VAR_IN_OUT PERSISTENT
	DsStnSeqRepCall : DSV2_fbStationSequenceRecipeCall;
	DsStnSubRepCall : DS_fbStationSubRecipeCall;
	DsBasketInfo : DSV2_BasketInfo;
END_VAR

VAR_OUTPUT PERSISTENT
	bProcessCompleted : BOOL;
	bProcessInProgressFlag : BOOL;
	bProcessHaltFlag: BOOL;
	bCallStnSeqRecipeErr: BOOL;
	bInvalidProcessStepErr: BOOL;
	DSStnSeqProOutput :DS_StnSeqProOutput;
	iCurrentProcessStep : INT;
	iComConProcessTimeEV: INT;
	ARiCurrentCycle : ARRAY [1..10] OF INT;
	iCurrentProcessTime : INT; (*Total Process Time Since Start*)
	iPreviousProcessTime : INT; (*Total Process Time - Previous process*)
	iStnSeqProcessCase: INT; (* Temporary - Will transfer to Var_Persistent later*)

END_VAR
VAR
(*	DsBufferSubRecipeMemory : Ds_SubRecipeMemory;
	bCallStnSeqSubProCompleted : BOOL;
	bCallStnSeqRepErr : BOOL;
	bCallStnSubRepErr : BOOL;
*)	rebProcessStart: R_TRIG;


	bCallStnSeqSubProEn: BOOL;

	bStCon7BelowTargetVacuumLevel : BOOL;
	bStCon8AboveTargetVacuumLevel : BOOL;
	bStCon9BelowTargetPressureLevel : BOOL;
	bStCon10AboveTargetPressureLevel : BOOL;
	bStCon11BelowTargetProTankTempLevel : BOOL;
	bStCon12AboveTargetProTankTempLevel : BOOL;
	bStCon13BelowTargetSubTankTempLevel : BOOL;
	bStCon14AboveTargetSubTankTempLevel : BOOL;

	bComCon7BelowTargetVacuumLevel : BOOL;
	bComCon8AboveTargetVacuumLevel : BOOL;
	bComCon9BelowTargetPressureLevel : BOOL;
	bComCon10AboveTargetPressureLevel : BOOL;
	bComCon11BelowTargetProTankTempLevel : BOOL;
	bComCon12AboveTargetProTankTempLevel : BOOL;
	bComCon13BelowTargetSubTankTempLevel : BOOL;
	bComCon14AboveTargetSubTankTempLevel : BOOL;

	tProcess1secClockPulse: TON;
	retProcess1secClockPulse: R_TRIG;
	rebProcessCompleted: R_TRIG;
	ClearFL: INT;
	iCurrentProcessStepBuffer: INT;
	rebInvalidProcessStepErr: R_TRIG;
	rebStnSeqSubCallCompleted: R_TRIG;
	rebCallStnSeqRecipeErr: R_TRIG;
	rebCallStnSubRecipeErr: R_TRIG;
	tStartProcess1secClockPulse: TON;
	retStartProcess1secClockPulse: R_TRIG;
	bTempCallCompleted: BOOL;
	bTempInvalidProcessStepErr: BOOL;
	bTempCallStnSeqRecipeErr: BOOL;
	bTempCallStnSubRecipeErr: BOOL;
	sTempsSubDescription: STRING(50);
	DsTempSubRecipeMemory: DS_SubRecipeMemory;
	iTempSeqStep: INT;
	bTempInvalidProcessStepErrPls: BOOL;
	rebProcessHalt: R_TRIG;
	febProcessHalt: F_TRIG;
END_VAR

VAR PERSISTENT
	StationfbCallStnSeqSubPro: fbCallStnSeqSubPro;
	bStartConditionPassed: BOOL;
	bCompleteConditionPassed: BOOL;
	bStationProcessTimerComplete: BOOL;
	iComConProcessTime: INT;

END_VAR

VAR_OUTPUT
END_VAR
*)

(*Temporary - Create Total Process Time SV *)
iTPTFL := 1;
bEndStep:= FALSE;

	FOR iTPTFL := 1 TO IStationSubRecipeArrayQty DO
		IF
		fbStationSequenceRecipefb.ARDsStorageStationSequenceRecipeMemory[DsBasketInfo.iStationSeqenceRecipeNo].AR10iStationSubProNo[iTPTFL] > 0
		AND
		fbStationSequenceRecipefb.ARDsStorageStationSequenceRecipeMemory[DsBasketInfo.iStationSeqenceRecipeNo].AR10iStationSubProNo[iTPTFL] <= IStationSubRecipeArrayQty
		AND NOT
		bEndStep
		THEN
		ARiTotalTimeSV[iTPTFL] := fbStationSubRecipefb.ARDsStorageSubRecipeMemory[(**)fbStationSequenceRecipefb.ARDsStorageStationSequenceRecipeMemory[DsBasketInfo.iStationSeqenceRecipeNo].AR10iStationSubProNo[iTPTFL](**)].iComCon5ProcessTimer;
		ELSE
		bEndStep := TRUE;
		ARiTotalTimeSV[iTPTFL] := 0;
		END_IF
	END_FOR
DsBasketInfo.iStationSeqenceRecipeNo;


iTotalProcessTimeSV :=
ARiTotalTimeSV[1] +
ARiTotalTimeSV[2] +
ARiTotalTimeSV[3] +
ARiTotalTimeSV[4] +
ARiTotalTimeSV[5] +
ARiTotalTimeSV[6] +
ARiTotalTimeSV[7] +
ARiTotalTimeSV[8] +
ARiTotalTimeSV[9] +
ARiTotalTimeSV[10];


IF bProcessInProgressFlag AND NOT bProcessHalt AND retStartProcess1secClockPulse.Q  THEN
iTotalProcessTimeEVInt := iTotalProcessTimeEVInt+1;
END_IF

IF (bProcessInProgressFlag OR bProcessHalt OR bProcessCompleted) AND NOT bProcessHalt AND iTotalProcessTimeSV - iTotalProcessTimeEVInt > 0 THEN
iTotalProcessTimeEV := iTotalProcessTimeSV - iTotalProcessTimeEVInt;
END_IF

IF (bProcessInProgressFlag OR bProcessHalt OR bProcessCompleted) AND NOT bProcessHalt AND iTotalProcessTimeSV - iTotalProcessTimeEVInt <= 0 THEN
iTotalProcessTimeEV := 0;
END_IF

IF NOT bProcessInProgressFlag AND NOT  bProcessHalt AND NOT bProcessCompleted THEN
iTotalProcessTimeEV := iTotalProcessTimeSV;
END_IF






(*Temp Create to generate total time for Loaded In Basket. Used in Time Optimisation*)
iCallTotalTimeMFL := 1;
iCallTotalTimeSFL := 1;

IF iCallTotalTimeMFL >0 AND iCallTotalTimeMFL < 5+1 THEN

	FOR iCallTotalTimeMFL := 1 TO 5 DO

		iCallTotalTimeSFL := 1;
		bCallTotalTimeEndStep:= FALSE;

		IF iCallTotalTimeSFL >0 AND iCallTotalTimeSFL < IStationSubRecipeArrayQty+1 THEN
			FOR iCallTotalTimeSFL := 1 TO IStationSubRecipeArrayQty DO
				IF
				fbStationSequenceRecipefb.ARDsStorageStationSequenceRecipeMemory[AR5iCallTotalTimeRecipeNo[iCallTotalTimeMFL]].AR10iStationSubProNo[iCallTotalTimeSFL] > 0
				AND
				fbStationSequenceRecipefb.ARDsStorageStationSequenceRecipeMemory[AR5iCallTotalTimeRecipeNo[iCallTotalTimeMFL]].AR10iStationSubProNo[iCallTotalTimeSFL] <= IStationSubRecipeArrayQty
				AND NOT
				bCallTotalTimeEndStep
				THEN
				AR2SiTimeOptimiseTotalTimeSV[iCallTotalTimeMFL,iCallTotalTimeSFL] := fbStationSubRecipefb.ARDsStorageSubRecipeMemory[(**)fbStationSequenceRecipefb.ARDsStorageStationSequenceRecipeMemory[AR5iCallTotalTimeRecipeNo[iCallTotalTimeMFL]].AR10iStationSubProNo[iCallTotalTimeSFL](**)].iComCon5ProcessTimer;
				ELSE
				bCallTotalTimeEndStep := TRUE;
				AR2SiTimeOptimiseTotalTimeSV[iCallTotalTimeMFL,iCallTotalTimeSFL] := 0;
				END_IF
			END_FOR
		END_IF
	END_FOR
END_IF

iCalculateMFL := 1;


IF iCalculateMFL >0 AND iCalculateMFL < 5+1 THEN

	FOR iCalculateMFL := 1 TO 5 DO

		AR5iCalledTotalProcessTimeSV[iCalculateMFL] :=
		AR2SiTimeOptimiseTotalTimeSV[iCalculateMFL,1] +
		AR2SiTimeOptimiseTotalTimeSV[iCalculateMFL,2] +
		AR2SiTimeOptimiseTotalTimeSV[iCalculateMFL,3] +
		AR2SiTimeOptimiseTotalTimeSV[iCalculateMFL,4] +
		AR2SiTimeOptimiseTotalTimeSV[iCalculateMFL,5] +
		AR2SiTimeOptimiseTotalTimeSV[iCalculateMFL,6] +
		AR2SiTimeOptimiseTotalTimeSV[iCalculateMFL,7] +
		AR2SiTimeOptimiseTotalTimeSV[iCalculateMFL,8] +
		AR2SiTimeOptimiseTotalTimeSV[iCalculateMFL,9] +
		AR2SiTimeOptimiseTotalTimeSV[iCalculateMFL,10];
		
	END_FOR
END_IF


(*[][][][][][][][][][][][][][][][][][][][][][][][][][][][][][][][][][][][][][][][][][][][][][][][][][][][][][][][][][][][][][][][][][][][][][][][]-Group in StationSequnceRecipe and StationSubRecipe-[][][][][][][][][][][][][][][][][][][][][][][][][][][][][][][][][][][][][][][][][][][][][][][][][][][][][][][][][][][][][][][][][][][][][][][][]*)
fbStationSequenceRecipefb(
	bSavePB								:=bSavePB ,
	bLoadPB								:=bLoadPB ,
	bClearPB							:=bClearPB_SSER ,
	bCopyPB								:=DsStnSeqRepStore.bCopyPB ,
	iCopyToSubRecipeNo						:=DsStnSeqRepStore.iCopyToSubRecipeNo ,
	iStnID									:=iCurrentStationAddress ,
	iStationSequenceRecipeNo				:=DsStnSeqRepStore.iStationSequenceRecipeNo ,
	sStationSequenceRecipeDescription			:=DsStnSeqRepStore.sStationSequenceRecipeDescription ,
	DsInStationSequenceRecipeMemory			:=DsStnSeqRepStore.DsStationSequenceRecipeMemory ,
	ARDsSSERSourceMinMaxTime_Uni			:=ARDsSSERSourceMinMaxTime_Uni ,
	Call_iStationSequenceRecipe				:=DsStnSeqRepCall.Call_iStationSequenceRecipe ,
	bCallPB									:=DsStnSeqRepCall.bCallPB ,
	bSaveInd								=>bSaveInd ,
	bLoadInd								=>bLoadInd ,
	bClearInd								=>bClearInd_SSUR ,
	bCallCompleted							=>DsStnSeqRepCall.bCallCompleted ,
	bInvalidCallStationSequenceNoHold			=>DsStnSeqRepCall.bInvalidCallStationSequenceNoHold ,
	bInvalidCallStationSequenceNoPulse		=>DsStnSeqRepCall.bInvalidCallStationSequenceNoPulse ,
	Call_sSequenceRecipeDescription			=>DsStnSeqRepCall.Call_sSequenceRecipeDescription ,
	Call_DsStationSequenceRecipeMemory		=>DsStnSeqRepCall.Call_DsStationSequenceRecipeMemory );

	

	
	
(*

fbStationSequenceRecipefb(
	bSavePB:=bSavePB ,
	bLoadPB:=bLoadPB ,
	bCopyPB:=DsStnSeqRepStore.bCopyPB ,
	iCopyToSubRecipeNo:= DsStnSeqRepStore.iCopyToSubRecipeNo,
	iStationSequenceRecipeNo:=DsStnSeqRepStore.iStationSequenceRecipeNo ,
	sStationSequenceRecipeDescription:=DsStnSeqRepStore.sStationSequenceRecipeDescription ,
	DsInStationSequenceRecipeMemory:=DsStnSeqRepStore.DsStationSequenceRecipeMemory ,
	Call_iStationSequenceRecipe:= DsStnSeqRepCall.Call_iStationSequenceRecipe,
	bCallPB:=DsStnSeqRepCall.bCallPB ,
	bSaveInd=>bSaveInd ,
	bLoadInd=>bLoadInd ,
	bCallCompleted=>DsStnSeqRepCall.bCallCompleted ,
	bInvalidCallStationSequenceNoHold=>DsStnSeqRepCall.bInvalidCallStationSequenceNoHold ,
	bInvalidCallStationSequenceNoPulse=>DsStnSeqRepCall.bInvalidCallStationSequenceNoPulse ,
	Call_sSequenceRecipeDescription=>DsStnSeqRepCall.Call_sSequenceRecipeDescription ,
	Call_DsStationSequenceRecipeMemory=>DsStnSeqRepCall.Call_DsStationSequenceRecipeMemory );
*)
fbStationSubRecipefb(
	bSavePB:= bSavePB,
	bLoadPB := bLoadPB,
	bClearPB:= bClearPB_SSUR,
	bCopyPB:=DsStnSubRepStore.bCopyPB ,
	iCopyToSubRecipeNo:= DsStnSubRepStore.iCopyToSubRecipeNo,
	DsStnSeqProInput:= DsStnSeqProInput,
	iSubRecipeNo:= DsStnSubRepStore.iSubRecipeNo,
	sSubRecipeDescription:= DsStnSubRepStore.sSubRecipeDescription,
	DsInSubRecipeMemory:= DsStnSubRepStore.DsSubRecipeMemory,
	Call_iSubRecipe:= DsStnSubRepCall.Call_iSubRecipe,
	bCallPB:= DsStnSubRepCall.bCallPB,
	bSaveInd=>bSaveInd ,
	bLoadInd=>bLoadInd ,
	bClearInd=>bClearInd_SSUR,
	bCallCompleted=> DsStnSubRepCall.bCallCompleted,
	bInvalidCallSubRecipeNoHold=> DsStnSubRepCall.bInvalidCallSubRecipeNoHold,
	bInvalidCallSubRecipeNoPulse=> DsStnSubRepCall.bInvalidCallSubRecipeNoPulse,
	Call_sSubDescription=> DsStnSubRepCall.Call_sSubDescription,
	Call_DsSubRecipeMemory=> DsStnSubRepCall.Call_DsSubRecipeMemory);


(*[][][][][][][][][][][][][][][][][][][][][][][][][][][][][][][][][][][][][][][][][][][][][][][][][][][][][][][][][][][][][][][][][][][][][][][][]-Only FB StnSeqProcess-[][][][][][][][][][][][][][][][][][][][][][][][][][][][][][][][][][][][][][][][][][][][][][][][][][][][][][][][][][][][][][][][][][][][][][][][]*)

(*[][][][][][][][][][][][][][][][][][]-Generate Current Process Time-[][][][][][][][][][][][][][][][][][]*)
tProcess1secClockPulse(IN:=(bProcessInProgressFlag OR bProcessCompleted) AND NOT tProcess1secClockPulse.Q , PT:= T#1s, Q=> , ET=> );
retProcess1secClockPulse(CLK:=tProcess1secClockPulse.Q , Q=> );

IF bProcessInProgressFlag AND NOT bProcessHalt AND retProcess1secClockPulse.Q THEN
iCurrentProcessTime := iCurrentProcessTime+1;
END_IF


IF (bProcessInProgressFlag OR bProcessCompleted OR bOutputCutOffEn) AND NOT bProcessHalt AND retProcess1secClockPulse.Q THEN
iNonStopCurrentProcessTime := iNonStopCurrentProcessTime+1;
END_IF


(*[][][][][][][][][][][][][][][][][][]-Complete Condition Process Time Handling-[][][][][][][][][][][][][][][][][][]*)

(*Generate CompleteCondition Process Time Elapse Value (Reverse Counting)*)
IF bProcessInProgressFlag AND NOT bProcessHalt AND StationfbCallStnSeqSubPro.BufferDsSubRecipeMemory.bComCon20EnProcessTimer AND iStnSeqProcessCaseNo = 3 THEN
iComConProcessTimeEV := StationfbCallStnSeqSubPro.BufferDsSubRecipeMemory.iComCon5ProcessTimer - iComConProcessTime;
END_IF

IF (NOT bProcessInProgressFlag AND NOT bProcessHalt) OR NOT StationfbCallStnSeqSubPro.BufferDsSubRecipeMemory.bComCon20EnProcessTimer OR iStnSeqProcessCaseNo <> 3 THEN
iComConProcessTimeEV := 0;
END_IF



(*Start Complete Condition Timer If Available*)
tStartProcess1secClockPulse(IN:=StationfbCallStnSeqSubPro.BufferDsSubRecipeMemory.bComCon20EnProcessTimer AND NOT tStartProcess1secClockPulse.Q AND iStnSeqProcessCaseNo = 3 , PT:=T#1s , Q=> , ET=> );
retStartProcess1secClockPulse(CLK:=tStartProcess1secClockPulse.Q , Q=> );

IF bProcessInProgressFlag AND NOT bProcessHalt AND retStartProcess1secClockPulse.Q  THEN
iComConProcessTime := iComConProcessTime+1;
END_IF

IF bProcessInProgressFlag AND NOT bProcessHalt AND iComConProcessTime >= StationfbCallStnSeqSubPro.BufferDsSubRecipeMemory.iComCon5ProcessTimer THEN
bStationProcessTimerComplete := TRUE;
ELSE
bStationProcessTimerComplete := FALSE;
END_IF


(*[][][][][][][][][][][][][][][][][][]-Generate Above/Below-Start Condition-[][][][][][][][][][][][][][][][][][]*)

IF DsStnSeqProInput.iVacuumLevelPV < StationfbCallStnSeqSubPro.BufferDsSubRecipeMemory.iStCon1TargetVacuumLevel THEN
bStCon11BelowTargetVacuumLevel := TRUE;
ELSE
bStCon11BelowTargetVacuumLevel := FALSE;
END_IF

IF DsStnSeqProInput.iVacuumLevelPV >= StationfbCallStnSeqSubPro.BufferDsSubRecipeMemory.iStCon1TargetVacuumLevel THEN
bStCon12AboveTargetVacuumLevel := TRUE;
ELSE
bStCon12AboveTargetVacuumLevel := FALSE;
END_IF

IF DsStnSeqProInput.iPressureLevelPV < StationfbCallStnSeqSubPro.BufferDsSubRecipeMemory.iStCon2TargetPressureLevel THEN
bStCon13BelowTargetPressureLevel := TRUE;
ELSE
bStCon13BelowTargetPressureLevel := FALSE;
END_IF

IF DsStnSeqProInput.iPressureLevelPV >= StationfbCallStnSeqSubPro.BufferDsSubRecipeMemory.iStCon2TargetPressureLevel THEN
bStCon14AboveTargetPressureLevel := TRUE;
ELSE
bStCon14AboveTargetPressureLevel := FALSE;
END_IF

IF DsStnSeqProInput.iProTankTempLevelPV < StationfbCallStnSeqSubPro.BufferDsSubRecipeMemory.iStCon3TargetProTankTempLevel THEN
bStCon15BelowTargetProTankTempLevel := TRUE;
ELSE
bStCon15BelowTargetProTankTempLevel := FALSE;
END_IF

IF DsStnSeqProInput.iProTankTempLevelPV >= StationfbCallStnSeqSubPro.BufferDsSubRecipeMemory.iStCon3TargetProTankTempLevel THEN
bStCon16AboveTargetProTankTempLevel := TRUE;
ELSE
bStCon16AboveTargetProTankTempLevel := FALSE;
END_IF

IF DsStnSeqProInput.iSubTankTempLevelPV < StationfbCallStnSeqSubPro.BufferDsSubRecipeMemory.iStCon4TargetSubTankTempLevel THEN
bStCon17BelowTargetSubTankTempLevel := TRUE;
ELSE
bStCon17BelowTargetSubTankTempLevel := FALSE;
END_IF

IF DsStnSeqProInput.iSubTankTempLevelPV >= StationfbCallStnSeqSubPro.BufferDsSubRecipeMemory.iStCon4TargetSubTankTempLevel THEN
bStCon18AboveTargetSubTankTempLevel := TRUE;
ELSE
bStCon18AboveTargetSubTankTempLevel := FALSE;
END_IF


(*[][][][][][][][][][][][][][][][][][]-Generate Above/Below-Complete Condition-[][][][][][][][][][][][][][][][][][]*)

IF DsStnSeqProInput.iVacuumLevelPV < StationfbCallStnSeqSubPro.BufferDsSubRecipeMemory.iComCon1TargetVacuumLevel THEN
bComCon11BelowTargetVacuumLevel := TRUE;
ELSE
bComCon11BelowTargetVacuumLevel := FALSE;
END_IF

IF DsStnSeqProInput.iVacuumLevelPV >= StationfbCallStnSeqSubPro.BufferDsSubRecipeMemory.iComCon1TargetVacuumLevel THEN
bComCon12AboveTargetVacuumLevel := TRUE;
ELSE
bComCon12AboveTargetVacuumLevel := FALSE;
END_IF

IF DsStnSeqProInput.iPressureLevelPV < StationfbCallStnSeqSubPro.BufferDsSubRecipeMemory.iComCon2TargetPressureLevel THEN
bComCon13BelowTargetPressureLevel := TRUE;
ELSE
bComCon13BelowTargetPressureLevel := FALSE;
END_IF

IF DsStnSeqProInput.iPressureLevelPV >= StationfbCallStnSeqSubPro.BufferDsSubRecipeMemory.iComCon2TargetPressureLevel THEN
bComCon14AboveTargetPressureLevel := TRUE;
ELSE
bComCon14AboveTargetPressureLevel := FALSE;
END_IF

IF DsStnSeqProInput.iProTankTempLevelPV < StationfbCallStnSeqSubPro.BufferDsSubRecipeMemory.iComCon3TargetProTankTempLevel THEN
bComCon15BelowTargetProTankTempLevel := TRUE;
ELSE
bComCon15BelowTargetProTankTempLevel := FALSE;
END_IF

IF DsStnSeqProInput.iProTankTempLevelPV >= StationfbCallStnSeqSubPro.BufferDsSubRecipeMemory.iComCon3TargetProTankTempLevel THEN
bComCon16AboveTargetProTankTempLevel := TRUE;
ELSE
bComCon16AboveTargetProTankTempLevel := FALSE;
END_IF

IF DsStnSeqProInput.iSubTankTempLevelPV < StationfbCallStnSeqSubPro.BufferDsSubRecipeMemory.iComCon4TargetSubTankTempLevel THEN
bComCon17BelowTargetSubTankTempLevel := TRUE;
ELSE
bComCon17BelowTargetSubTankTempLevel := FALSE;
END_IF

IF DsStnSeqProInput.iSubTankTempLevelPV >= StationfbCallStnSeqSubPro.BufferDsSubRecipeMemory.iComCon4TargetSubTankTempLevel THEN
bComCon18AboveTargetSubTankTempLevel := TRUE;
ELSE
bComCon18AboveTargetSubTankTempLevel := FALSE;
END_IF

(*[][][][][][][][][][][][][][][][][][]-General-[][][][][][][][][][][][][][][][][][]*)
rebProcessHalt(CLK:=bProcessHalt , Q=> );

febProcessHalt(CLK:=bProcessHalt , Q=> );

IF rebProcessHalt.Q AND bProcessInProgressFlag THEN
bProcessInProgressFlag := FALSE;
bProcessHaltFlag := TRUE;
END_IF

IF febProcessHalt.Q AND bProcessHaltFlag THEN
bProcessInProgressFlag := TRUE;
bProcessHaltFlag := FALSE;
END_IF



IF bProcessReset OR NOT DsBasketInfo.bAvailibility THEN
bProcessInProgressFlag := FALSE;
bCallStnSeqRecipeErr := FALSE;
bInvalidProcessStepErr := FALSE;
bCallStnSeqSubProEn := FALSE;
bProcessCompleted := FALSE;
bProcessHaltFlag := FALSE;

iStnSeqProcessCaseNo := 0;
iCurrentProcessStep := 0;
iCurrentProcessTime := 0;
iNonStopCurrentProcessTime := 0;
(*iTotalProcessTimeEV:=0;*)
iTotalProcessTimeEVInt := 0;
iComConProcessTime := 0;
iTotalProcessTimeEV := 0; (*Add New*)
DsStnSeqRepCall:=DsStnSeqRepCallEmpty;
DsStnSubRepCall:=DsStnSubRepCallEmpty;
ClearFL := 1;

	FOR ClearFL := 1 TO IStationSubRecipeArrayQty(*10*) DO
		ARiCurrentCycle[ClearFL] := 0;
	END_FOR

END_IF




rebProcessStart(CLK:=bProcessStart  , Q=> );

IF rebProcessStart.Q AND NOT bProcessHaltFlag AND NOT bProcessInProgressFlag AND NOT bProcessCompleted THEN
iStnSeqProcessCaseNo := 1;
iCurrentProcessStep := 1;
ARiCurrentCycle[iCurrentProcessStep] := 1;
bProcessInProgressFlag := TRUE;
END_IF


(*[][][][][][][][][][][][][][][][][][]-FB Declaration-[][][][][][][][][][][][][][][][][][]*)

StationfbCallStnSeqSubPro(
	bCallSt:= bCallStnSeqSubProEn ,
	iCurrentProcessStep:=iCurrentProcessStep ,
	DSStnSeqRepCall:=DsStnSeqRepCall ,
	DSStnSeqSubCall:=DsStnSubRepCall ,
	DSBasketInfo:=DsBasketInfo ,
	bCallCompleted=>bTempCallCompleted ,
	bInvalidProcessStepErrHold=>bTempInvalidProcessStepErr ,
	bInvalidProcessStepErrPulse=>bTempInvalidProcessStepErrPls,
	bCallStnSeqRecipeErr=> bTempCallStnSeqRecipeErr,
	bCallStnSubRecipeErr=> bTempCallStnSubRecipeErr,
	BuffersSubDescription=> sTempsSubDescription,
	BufferDsSubRecipeMemory=> DsTempSubRecipeMemory,
	iSeqStep=> iTempSeqStep);


(*[][][][][][][][][][][][][][][][][][]-Main-Case/Step Programming-[][][][][][][][][][][][][][][][][][]*)

rebStnSeqSubCallCompleted(CLK:=StationfbCallStnSeqSubPro.bCallCompleted , Q=> );
rebCallStnSeqRecipeErr(CLK:=StationfbCallStnSeqSubPro.bCallStnSeqRecipeErr , Q=> );
rebInvalidProcessStepErr(CLK:=StationfbCallStnSeqSubPro.bInvalidProcessStepErrPulse , Q=> );
rebCallStnSubRecipeErr(CLK:=StationfbCallStnSeqSubPro.bCallStnSubRecipeErr , Q=> );


CASE iStnSeqProcessCaseNo OF

0:;

1: (*Pull Data from fbCallStnSeqSubPro*)
bCallStnSeqSubProEn:= TRUE;

IF rebStnSeqSubCallCompleted.Q THEN
bCallStnSeqSubProEn := FALSE;
bStartConditionPassed := FALSE;
bCompleteConditionPassed := FALSE;
iStnSeqProcessCaseNo := 2;
END_IF

IF rebCallStnSeqRecipeErr.Q THEN
bCallStnSeqSubProEn := FALSE;
bStartConditionPassed := FALSE;
bCompleteConditionPassed := FALSE;
iStnSeqProcessCaseNo := 90;
END_IF

IF rebInvalidProcessStepErr.Q THEN
bCallStnSeqSubProEn := FALSE;
bStartConditionPassed := FALSE;
bCompleteConditionPassed := FALSE;
iStnSeqProcessCaseNo := 91;
END_IF

IF rebCallStnSubRecipeErr.Q THEN
bCallStnSeqSubProEn := FALSE;
bStartConditionPassed := FALSE;
bCompleteConditionPassed := FALSE;
iStnSeqProcessCaseNo := 92;
END_IF

2: (*Start Condition Validation*)
IF bProcessInProgressFlag AND (
(StationfbCallStnSeqSubPro.BufferDsSubRecipeMemory.bStCon1EnProLowLiquidLevel AND NOT DsStnSeqProInput.bProLowLiquidLevel_NC) OR
(StationfbCallStnSeqSubPro.BufferDsSubRecipeMemory.bStCon2EnProRegLiquidLevel AND DsStnSeqProInput.bProRegLiquidLevel_NO) OR
(StationfbCallStnSeqSubPro.BufferDsSubRecipeMemory.bStCon3EnProHighLiquidLevel AND DsStnSeqProInput.bProHighLiquidLevel_NO) OR
(StationfbCallStnSeqSubPro.BufferDsSubRecipeMemory.bStCon4EnSubLowLiquidLevel AND NOT DsStnSeqProInput.bSubLowLiquidLevel_NC) OR
(StationfbCallStnSeqSubPro.BufferDsSubRecipeMemory.bStCon5EnSubRegLiquidLevel AND DsStnSeqProInput.bSubRegLiquidLevel_NO) OR
(StationfbCallStnSeqSubPro.BufferDsSubRecipeMemory.bStCon6EnSubHighLiquidLevel AND DsStnSeqProInput.bSubHighLiquidLevel_NO) OR

(StationfbCallStnSeqSubPro.BufferDsSubRecipeMemory.bStCon7EnLowVacuumLevel AND DsStnSeqProInput.bLowVacuumLevel_NO) OR
(StationfbCallStnSeqSubPro.BufferDsSubRecipeMemory.bStCon8EnRegVacuumLevel AND DsStnSeqProInput.bRegVacuumLevel_NO) OR
(StationfbCallStnSeqSubPro.BufferDsSubRecipeMemory.bStCon9EnLowPressureLevel AND DsStnSeqProInput.bLowPressureLevel_NO) OR
(StationfbCallStnSeqSubPro.BufferDsSubRecipeMemory.bStCon10EnRegPressureLevel AND DsStnSeqProInput.bRegPressureLevel_NO) OR
(StationfbCallStnSeqSubPro.BufferDsSubRecipeMemory.bStCon11EnBelowTargetVacuumLevel AND bStCon11BelowTargetVacuumLevel) OR
(StationfbCallStnSeqSubPro.BufferDsSubRecipeMemory.bStCon12EnAboveTargetVacuumLevel AND bStCon12AboveTargetVacuumLevel) OR
(StationfbCallStnSeqSubPro.BufferDsSubRecipeMemory.bStCon13EnBelowTargetPressureLevel AND bStCon13BelowTargetPressureLevel) OR
(StationfbCallStnSeqSubPro.BufferDsSubRecipeMemory.bStCon14EnAboveTargetPressureLevel AND bStCon14AboveTargetPressureLevel) OR
(StationfbCallStnSeqSubPro.BufferDsSubRecipeMemory.bStCon15EnBelowTargetProTankTempLevel AND bStCon15BelowTargetProTankTempLevel) OR
(StationfbCallStnSeqSubPro.BufferDsSubRecipeMemory.bStCon16EnAboveTargetProTankTempLevel AND bStCon16AboveTargetProTankTempLevel) OR
(StationfbCallStnSeqSubPro.BufferDsSubRecipeMemory.bStCon17EnBelowTargetSubTankTempLevel AND bStCon17BelowTargetSubTankTempLevel) OR
(StationfbCallStnSeqSubPro.BufferDsSubRecipeMemory.bStCon18EnAboveTargetSubTankTempLevel AND bStCon18AboveTargetSubTankTempLevel) OR
(StationfbCallStnSeqSubPro.BufferDsSubRecipeMemory.bStCon19ExternalActivation AND DsStnSeqProInput.bExternalActivation_NO) OR

(NOT StationfbCallStnSeqSubPro.BufferDsSubRecipeMemory.bStCon1EnProLowLiquidLevel
AND NOT StationfbCallStnSeqSubPro.BufferDsSubRecipeMemory.bStCon2EnProRegLiquidLevel
AND NOT StationfbCallStnSeqSubPro.BufferDsSubRecipeMemory.bStCon3EnProHighLiquidLevel
AND NOT StationfbCallStnSeqSubPro.BufferDsSubRecipeMemory.bStCon4EnSubLowLiquidLevel
AND NOT StationfbCallStnSeqSubPro.BufferDsSubRecipeMemory.bStCon5EnSubRegLiquidLevel
AND NOT StationfbCallStnSeqSubPro.BufferDsSubRecipeMemory.bStCon6EnSubHighLiquidLevel

AND NOT StationfbCallStnSeqSubPro.BufferDsSubRecipeMemory.bStCon7EnLowVacuumLevel
AND NOT StationfbCallStnSeqSubPro.BufferDsSubRecipeMemory.bStCon8EnRegVacuumLevel
AND NOT StationfbCallStnSeqSubPro.BufferDsSubRecipeMemory.bStCon9EnLowPressureLevel
AND NOT StationfbCallStnSeqSubPro.BufferDsSubRecipeMemory.bStCon10EnRegPressureLevel
AND NOT StationfbCallStnSeqSubPro.BufferDsSubRecipeMemory.bStCon11EnBelowTargetVacuumLevel
AND NOT StationfbCallStnSeqSubPro.BufferDsSubRecipeMemory.bStCon12EnAboveTargetVacuumLevel
AND NOT StationfbCallStnSeqSubPro.BufferDsSubRecipeMemory.bStCon13EnBelowTargetPressureLevel
AND NOT StationfbCallStnSeqSubPro.BufferDsSubRecipeMemory.bStCon14EnAboveTargetPressureLevel
AND NOT StationfbCallStnSeqSubPro.BufferDsSubRecipeMemory.bStCon15EnBelowTargetProTankTempLevel
AND NOT StationfbCallStnSeqSubPro.BufferDsSubRecipeMemory.bStCon16EnAboveTargetProTankTempLevel
AND NOT StationfbCallStnSeqSubPro.BufferDsSubRecipeMemory.bStCon17EnBelowTargetSubTankTempLevel
AND NOT StationfbCallStnSeqSubPro.BufferDsSubRecipeMemory.bStCon18EnAboveTargetSubTankTempLevel
AND NOT StationfbCallStnSeqSubPro.BufferDsSubRecipeMemory.bStCon19ExternalActivation) )THEN

bStartConditionPassed := TRUE;
iStnSeqProcessCaseNo := 3;
END_IF

3: (* Process Start Progress and Waiting Validate Complete Condition*)



(*Complete Condition Validation*)
IF bProcessInProgressFlag AND (
(StationfbCallStnSeqSubPro.BufferDsSubRecipeMemory.bComCon1EnProLowLiquidLevel AND NOT DsStnSeqProInput.bProLowLiquidLevel_NC) OR
(StationfbCallStnSeqSubPro.BufferDsSubRecipeMemory.bComCon2EnProRegLiquidLevel AND DsStnSeqProInput.bProRegLiquidLevel_NO) OR
(StationfbCallStnSeqSubPro.BufferDsSubRecipeMemory.bComCon3EnProHighLiquidLevel AND DsStnSeqProInput.bProHighLiquidLevel_NO) OR
(StationfbCallStnSeqSubPro.BufferDsSubRecipeMemory.bComCon4EnSubLowLiquidLevel AND NOT DsStnSeqProInput.bSubLowLiquidLevel_NC) OR
(StationfbCallStnSeqSubPro.BufferDsSubRecipeMemory.bComCon5EnSubRegLiquidLevel AND DsStnSeqProInput.bSubRegLiquidLevel_NO) OR
(StationfbCallStnSeqSubPro.BufferDsSubRecipeMemory.bComCon6EnSubHighLiquidLevel AND DsStnSeqProInput.bSubHighLiquidLevel_NO) OR

(StationfbCallStnSeqSubPro.BufferDsSubRecipeMemory.bComCon7EnLowVacuumLevel AND DsStnSeqProInput.bLowVacuumLevel_NO) OR
(StationfbCallStnSeqSubPro.BufferDsSubRecipeMemory.bComCon8EnRegVacuumLevel AND DsStnSeqProInput.bRegVacuumLevel_NO) OR
(StationfbCallStnSeqSubPro.BufferDsSubRecipeMemory.bComCon9EnLowPressureLevel AND DsStnSeqProInput.bLowPressureLevel_NO) OR
(StationfbCallStnSeqSubPro.BufferDsSubRecipeMemory.bComCon10EnRegPressureLevel AND DsStnSeqProInput.bRegPressureLevel_NO) OR
(StationfbCallStnSeqSubPro.BufferDsSubRecipeMemory.bComCon11EnBelowTargetVacuumLevel AND bComCon11BelowTargetVacuumLevel) OR
(StationfbCallStnSeqSubPro.BufferDsSubRecipeMemory.bComCon12EnAboveTargetVacuumLevel AND bComCon12AboveTargetVacuumLevel) OR
(StationfbCallStnSeqSubPro.BufferDsSubRecipeMemory.bComCon13EnBelowTargetPressureLevel AND bComCon13BelowTargetPressureLevel) OR
(StationfbCallStnSeqSubPro.BufferDsSubRecipeMemory.bComCon14EnAboveTargetPressureLevel AND bComCon14AboveTargetPressureLevel) OR
(StationfbCallStnSeqSubPro.BufferDsSubRecipeMemory.bComCon15EnBelowTargetProTankTempLevel AND bComCon15BelowTargetProTankTempLevel) OR
(StationfbCallStnSeqSubPro.BufferDsSubRecipeMemory.bComCon16EnAboveTargetProTankTempLevel AND bComCon16AboveTargetProTankTempLevel) OR
(StationfbCallStnSeqSubPro.BufferDsSubRecipeMemory.bComCon17EnBelowTargetSubTankTempLevel AND bComCon17BelowTargetSubTankTempLevel) OR
(StationfbCallStnSeqSubPro.BufferDsSubRecipeMemory.bComCon18EnAboveTargetSubTankTempLevel AND bComCon18AboveTargetSubTankTempLevel) OR
(StationfbCallStnSeqSubPro.BufferDsSubRecipeMemory.bComCon19EnExternalActivation AND DsStnSeqProInput.bExternalActivation_NO) OR

(StationfbCallStnSeqSubPro.BufferDsSubRecipeMemory.bComCon20EnProcessTimer AND bStationProcessTimerComplete) OR

(NOT StationfbCallStnSeqSubPro.BufferDsSubRecipeMemory.bComCon1EnProLowLiquidLevel
AND NOT StationfbCallStnSeqSubPro.BufferDsSubRecipeMemory.bComCon2EnProRegLiquidLevel
AND NOT StationfbCallStnSeqSubPro.BufferDsSubRecipeMemory.bComCon3EnProHighLiquidLevel
AND NOT StationfbCallStnSeqSubPro.BufferDsSubRecipeMemory.bComCon4EnSubLowLiquidLevel
AND NOT StationfbCallStnSeqSubPro.BufferDsSubRecipeMemory.bComCon5EnSubRegLiquidLevel
AND NOT StationfbCallStnSeqSubPro.BufferDsSubRecipeMemory.bComCon6EnSubHighLiquidLevel
AND NOT StationfbCallStnSeqSubPro.BufferDsSubRecipeMemory.bComCon7EnLowVacuumLevel
AND NOT StationfbCallStnSeqSubPro.BufferDsSubRecipeMemory.bComCon8EnRegVacuumLevel
AND NOT StationfbCallStnSeqSubPro.BufferDsSubRecipeMemory.bComCon9EnLowPressureLevel
AND NOT StationfbCallStnSeqSubPro.BufferDsSubRecipeMemory.bComCon10EnRegPressureLevel
AND NOT StationfbCallStnSeqSubPro.BufferDsSubRecipeMemory.bComCon11EnBelowTargetVacuumLevel
AND NOT StationfbCallStnSeqSubPro.BufferDsSubRecipeMemory.bComCon12EnAboveTargetVacuumLevel
AND NOT StationfbCallStnSeqSubPro.BufferDsSubRecipeMemory.bComCon13EnBelowTargetPressureLevel
AND NOT StationfbCallStnSeqSubPro.BufferDsSubRecipeMemory.bComCon14EnAboveTargetPressureLevel
AND NOT StationfbCallStnSeqSubPro.BufferDsSubRecipeMemory.bComCon15EnBelowTargetProTankTempLevel
AND NOT StationfbCallStnSeqSubPro.BufferDsSubRecipeMemory.bComCon16EnAboveTargetProTankTempLevel
AND NOT StationfbCallStnSeqSubPro.BufferDsSubRecipeMemory.bComCon17EnBelowTargetSubTankTempLevel
AND NOT StationfbCallStnSeqSubPro.BufferDsSubRecipeMemory.bComCon18EnAboveTargetSubTankTempLevel
AND NOT StationfbCallStnSeqSubPro.BufferDsSubRecipeMemory.bComCon19EnExternalActivation
AND NOT StationfbCallStnSeqSubPro.BufferDsSubRecipeMemory.bComCon20EnProcessTimer) )THEN

bCompleteConditionPassed := TRUE;
iStnSeqProcessCaseNo := 4;
END_IF


(*Trigger Output*)

IF bProcessInProgressFlag THEN
DSStnSeqProOutput.b1ProTankPump := StationfbCallStnSeqSubPro.BufferDsSubRecipeMemory.bOut1EnProTankPump;
DSStnSeqProOutput.b2ProTankHeater := StationfbCallStnSeqSubPro.BufferDsSubRecipeMemory.bOut2EnProTankHeater;
DSStnSeqProOutput.b3ProTankBottomUltrasonicA := StationfbCallStnSeqSubPro.BufferDsSubRecipeMemory.bOut3EnProTankBottomUltrasonicA;
DSStnSeqProOutput.b4ProTankBottomUltrasonicB := StationfbCallStnSeqSubPro.BufferDsSubRecipeMemory.bOut4EnProTankBottomUltrasonicB;
DSStnSeqProOutput.b5ProTankBottomUltrasonicC := StationfbCallStnSeqSubPro.BufferDsSubRecipeMemory.bOut5EnProTankBottomUltrasonicC;
DSStnSeqProOutput.b6ProTankSideUltrasonicA := StationfbCallStnSeqSubPro.BufferDsSubRecipeMemory.bOut6EnProTankSideUltrasonicA;
DSStnSeqProOutput.b7ProTankSideUltrasonicB := StationfbCallStnSeqSubPro.BufferDsSubRecipeMemory.bOut7EnProTankSideUltrasonicB;
DSStnSeqProOutput.b8SubTankPump := StationfbCallStnSeqSubPro.BufferDsSubRecipeMemory.bOut8EnSubTankPump;
DSStnSeqProOutput.b9SubTankHeater := StationfbCallStnSeqSubPro.BufferDsSubRecipeMemory.bOut9EnSubTankHeater;
DSStnSeqProOutput.b10Blower := StationfbCallStnSeqSubPro.BufferDsSubRecipeMemory.bOut10EnBlower;
DSStnSeqProOutput.b11VacuumPump := StationfbCallStnSeqSubPro.BufferDsSubRecipeMemory.bOut11EnVacuumPump;
DSStnSeqProOutput.b12SlowPull := StationfbCallStnSeqSubPro.BufferDsSubRecipeMemory.bOut12EnSlowPull;
DSStnSeqProOutput.b13Instrument2 := StationfbCallStnSeqSubPro.BufferDsSubRecipeMemory.bOut13EnInstrument2;
DSStnSeqProOutput.b14Instrument3 := StationfbCallStnSeqSubPro.BufferDsSubRecipeMemory.bOut14EnInstrument3;
DSStnSeqProOutput.b15Instrument4 := StationfbCallStnSeqSubPro.BufferDsSubRecipeMemory.bOut15EnInstrument4;

DSStnSeqProOutput.b16EnProTankChangeTemp := StationfbCallStnSeqSubPro.BufferDsSubRecipeMemory.bOut16EnProTankChangeTemperature;
DSStnSeqProOutput.b17EnSubTankChangeTemp := StationfbCallStnSeqSubPro.BufferDsSubRecipeMemory.bOut17EnSubTankChangeTemperature;

DSStnSeqProOutput.b1ActValve1 := StationfbCallStnSeqSubPro.BufferDsSubRecipeMemory.bOut1ActValve1;
DSStnSeqProOutput.b2ActValve2 := StationfbCallStnSeqSubPro.BufferDsSubRecipeMemory.bOut2ActValve2;
DSStnSeqProOutput.b3ActValve3 := StationfbCallStnSeqSubPro.BufferDsSubRecipeMemory.bOut3ActValve3;
DSStnSeqProOutput.b4ActValve4 := StationfbCallStnSeqSubPro.BufferDsSubRecipeMemory.bOut4ActValve4;
DSStnSeqProOutput.b5ActValve5 := StationfbCallStnSeqSubPro.BufferDsSubRecipeMemory.bOut5ActValve5;
DSStnSeqProOutput.b6ActValve6 := StationfbCallStnSeqSubPro.BufferDsSubRecipeMemory.bOut6ActValve6;
DSStnSeqProOutput.b7ActValve7 := StationfbCallStnSeqSubPro.BufferDsSubRecipeMemory.bOut7ActValve7;
DSStnSeqProOutput.b8ActValve8 := StationfbCallStnSeqSubPro.BufferDsSubRecipeMemory.bOut8ActValve8;
DSStnSeqProOutput.b9ActValve9 := StationfbCallStnSeqSubPro.BufferDsSubRecipeMemory.bOut9ActValve9;
DSStnSeqProOutput.b10ActValve10 := StationfbCallStnSeqSubPro.BufferDsSubRecipeMemory.bOut10ActValve10;
DSStnSeqProOutput.b11ActValve11 := StationfbCallStnSeqSubPro.BufferDsSubRecipeMemory.bOut11ActValve11;
DSStnSeqProOutput.b12ActValve12 := StationfbCallStnSeqSubPro.BufferDsSubRecipeMemory.bOut12ActValve12;
DSStnSeqProOutput.b13ActValve13 := StationfbCallStnSeqSubPro.BufferDsSubRecipeMemory.bOut13ActValve13;
DSStnSeqProOutput.b14ActValve14 := StationfbCallStnSeqSubPro.BufferDsSubRecipeMemory.bOut14ActValve14;
DSStnSeqProOutput.b15ActValve15 := StationfbCallStnSeqSubPro.BufferDsSubRecipeMemory.bOut15ActValve15;
DSStnSeqProOutput.b16ActValve16 := StationfbCallStnSeqSubPro.BufferDsSubRecipeMemory.bOut16ActValve16;
DSStnSeqProOutput.b17ActValve17 := StationfbCallStnSeqSubPro.BufferDsSubRecipeMemory.bOut17ActValve17;
DSStnSeqProOutput.b18ActValve18 := StationfbCallStnSeqSubPro.BufferDsSubRecipeMemory.bOut18ActValve18;
DSStnSeqProOutput.b19ActValve19 := StationfbCallStnSeqSubPro.BufferDsSubRecipeMemory.bOut19ActValve19;
DSStnSeqProOutput.b20ActValve20 := StationfbCallStnSeqSubPro.BufferDsSubRecipeMemory.bOut20ActValve20;

DSStnSeqProOutput.i1ProTankPumpLPM := StationfbCallStnSeqSubPro.BufferDsSubRecipeMemory.iOut1ProTankPumpLPM;
DSStnSeqProOutput.i2ProTankPumpHz := StationfbCallStnSeqSubPro.BufferDsSubRecipeMemory.iOut2ProTankPumpHz;
DSStnSeqProOutput.i3ProTankBtmUsAPwrPercent := StationfbCallStnSeqSubPro.BufferDsSubRecipeMemory.iOut3ProTankBtmUsAPwrPercent;
DSStnSeqProOutput.i4ProTankBtmUsBPwrPercent := StationfbCallStnSeqSubPro.BufferDsSubRecipeMemory.iOut4ProTankBtmUsBPwrPercent;
DSStnSeqProOutput.i5ProTankBtmUsCPwrPercent := StationfbCallStnSeqSubPro.BufferDsSubRecipeMemory.iOut5ProTankBtmUsCPwrPercent;
DSStnSeqProOutput.i6ProTankSideUsAPwrPercent := StationfbCallStnSeqSubPro.BufferDsSubRecipeMemory.iOut6ProTankSideUsAPwrPercent;
DSStnSeqProOutput.i7ProTankSideUsBPwrPercent := StationfbCallStnSeqSubPro.BufferDsSubRecipeMemory.iOut7ProTankSideUsBPwrPercent;
DSStnSeqProOutput.i8ProTankBtmUsAkHz := StationfbCallStnSeqSubPro.BufferDsSubRecipeMemory.iOut8ProTankBtmUsAkHz;
DSStnSeqProOutput.i9ProTankBtmUsBkHz := StationfbCallStnSeqSubPro.BufferDsSubRecipeMemory.iOut9ProTankBtmUsBkHz;
DSStnSeqProOutput.i10ProTankBtmUsCkHz := StationfbCallStnSeqSubPro.BufferDsSubRecipeMemory.iOut10ProTankBtmUsCkHz;
DSStnSeqProOutput.i11ProTankSideUsAkHz := StationfbCallStnSeqSubPro.BufferDsSubRecipeMemory.iOut11ProTankSideUsAkHz;
DSStnSeqProOutput.i12ProTankSideUsBkHz := StationfbCallStnSeqSubPro.BufferDsSubRecipeMemory.iOut12ProTankSideUsBkHz;
DSStnSeqProOutput.i13ProTankBlowerHz := StationfbCallStnSeqSubPro.BufferDsSubRecipeMemory.iOut13ProTankBlowerHz;
DSStnSeqProOutput.i16SubTankPumpLPM := StationfbCallStnSeqSubPro.BufferDsSubRecipeMemory.iOut16SubTankPumpLPM;
DSStnSeqProOutput.i17SubTankPumpHz := StationfbCallStnSeqSubPro.BufferDsSubRecipeMemory.iOut17SubTankPumpHz;

DSStnSeqProOutput.i18SlowPullVelocity := StationfbCallStnSeqSubPro.BufferDsSubRecipeMemory.iOut18SlowPullVelocity;

IF StationfbCallStnSeqSubPro.BufferDsSubRecipeMemory.iOut19SlowPullDelayTime - iComConProcessTime > 0 THEN
DSStnSeqProOutput.i19SlowPullDelayTime := StationfbCallStnSeqSubPro.BufferDsSubRecipeMemory.iOut19SlowPullDelayTime - iComConProcessTime;
ELSE
DSStnSeqProOutput.i19SlowPullDelayTime := 0;
END_IF




IF DSStnSeqProOutput.b16EnProTankChangeTemp THEN
	DSStnSeqProOutput.r14ProTankChangeTempDegC := StationfbCallStnSeqSubPro.BufferDsSubRecipeMemory.rOut14ProTankChangeTemperatureDegC;
ELSE
	DSStnSeqProOutput.r14ProTankChangeTempDegC := 0;
END_IF


IF DSStnSeqProOutput.b17EnSubTankChangeTemp THEN
	DSStnSeqProOutput.r15SubTankChangeTempDegC := StationfbCallStnSeqSubPro.BufferDsSubRecipeMemory.rOut15SubTankChangeTemperatureDegC;
ELSE
	DSStnSeqProOutput.r15SubTankChangeTempDegC := 0;
END_IF






END_IF


4: (* Repeat Sequence *)

IF ARiCurrentCycle[iCurrentProcessStep] >= DsStnSeqRepCall.Call_DsStationSequenceRecipeMemory.AR10iCycle[iCurrentProcessStep] THEN

ARiCurrentCycle[iCurrentProcessStep] := 0;
iCurrentProcessStep := iCurrentProcessStep+1;
ARiCurrentCycle[iCurrentProcessStep] := ARiCurrentCycle[iCurrentProcessStep]  +1;
iStnSeqProcessCaseNo := 6;

ELSE
iCurrentProcessStepBuffer :=DsStnSeqRepCall.Call_DsStationSequenceRecipeMemory.AR10iRepeatFromStepNo[iCurrentProcessStep];
iStnSeqProcessCaseNo := 5;
END_IF

5: (*Move CurrentProcessStepBuffer to CurrentProcessStep*)
iCurrentProcessStep := iCurrentProcessStepBuffer;
ARiCurrentCycle[iCurrentProcessStep] := ARiCurrentCycle[iCurrentProcessStep]  +1;
iStnSeqProcessCaseNo := 6;

6: (* Trigger Repeat Process*)
bStartConditionPassed := FALSE;
bCompleteConditionPassed := FALSE;
iComConProcessTime := 0;
iStnSeqProcessCaseNo := 1;

90:(*Trigger Call Station Sequence Recipe Error*);
bCallStnSeqRecipeErr := TRUE;
bProcessInProgressFlag := FALSE;
iStnSeqProcessCaseNo := 97;

91:(*Trigger Invalid Process Step Error*)
bInvalidProcessStepErr := TRUE;
bProcessInProgressFlag := FALSE;
iStnSeqProcessCaseNo := 98;

92: (*Trigger Process Complete Flag*)
bProcessCompleted := TRUE;
bProcessInProgressFlag := FALSE;
iPreviousProcessTime := iCurrentProcessTime;
iCurrentProcessTime := 0;
iStnSeqProcessCaseNo := 99;


97:(*Stay if Call Station Sequence Recipe Error*)
;
98:(*Stay if Invalid Process Step Error*)
;
99:(*Stay if Process Completed*)
;

END_CASE



(*[][][][][][][][][][][][][][][][][][]-Stop Output when Process is Stop/Complete/Halt-[][][][][][][][][][][][][][][][][][]*)

IF NOT bProcessInProgressFlag OR bOutputCutOffEn THEN
DSStnSeqProOutput.b1ProTankPump := FALSE;
DSStnSeqProOutput.b2ProTankHeater := FALSE;
DSStnSeqProOutput.b3ProTankBottomUltrasonicA := FALSE;
DSStnSeqProOutput.b4ProTankBottomUltrasonicB := FALSE;
DSStnSeqProOutput.b5ProTankBottomUltrasonicC := FALSE;
DSStnSeqProOutput.b6ProTankSideUltrasonicA := FALSE;
DSStnSeqProOutput.b7ProTankSideUltrasonicB := FALSE;
DSStnSeqProOutput.b8SubTankPump := FALSE;
DSStnSeqProOutput.b9SubTankHeater := FALSE;
DSStnSeqProOutput.b10Blower := FALSE;
DSStnSeqProOutput.b11VacuumPump := FALSE;
DSStnSeqProOutput.b12SlowPull := FALSE;
DSStnSeqProOutput.b13Instrument2 := FALSE;
DSStnSeqProOutput.b14Instrument3 := FALSE;
DSStnSeqProOutput.b15Instrument4 := FALSE;

DSStnSeqProOutput.b16EnProTankChangeTemp := FALSE;
DSStnSeqProOutput.b17EnSubTankChangeTemp := FALSE;



DSStnSeqProOutput.b1ActValve1 := FALSE;
DSStnSeqProOutput.b2ActValve2 := FALSE;
DSStnSeqProOutput.b3ActValve3 := FALSE;
DSStnSeqProOutput.b4ActValve4 := FALSE;
DSStnSeqProOutput.b5ActValve5 := FALSE;
DSStnSeqProOutput.b6ActValve6 := FALSE;
DSStnSeqProOutput.b7ActValve7 := FALSE;
DSStnSeqProOutput.b8ActValve8 := FALSE;
DSStnSeqProOutput.b9ActValve9 := FALSE;
DSStnSeqProOutput.b10ActValve10 := FALSE;
DSStnSeqProOutput.b11ActValve11 := FALSE;
DSStnSeqProOutput.b12ActValve12 := FALSE;
DSStnSeqProOutput.b13ActValve13 := FALSE;
DSStnSeqProOutput.b14ActValve14 := FALSE;
DSStnSeqProOutput.b15ActValve15 := FALSE;
DSStnSeqProOutput.b16ActValve16 := FALSE;
DSStnSeqProOutput.b17ActValve17 := FALSE;
DSStnSeqProOutput.b18ActValve18 := FALSE;
DSStnSeqProOutput.b19ActValve19 := FALSE;
DSStnSeqProOutput.b20ActValve20 := FALSE;

DSStnSeqProOutput.i1ProTankPumpLPM := 0;
DSStnSeqProOutput.i2ProTankPumpHz := 0;
DSStnSeqProOutput.i3ProTankBtmUsAPwrPercent := 0;
DSStnSeqProOutput.i4ProTankBtmUsBPwrPercent := 0;
DSStnSeqProOutput.i5ProTankBtmUsCPwrPercent := 0;
DSStnSeqProOutput.i6ProTankSideUsAPwrPercent := 0;
DSStnSeqProOutput.i7ProTankSideUsBPwrPercent := 0;
DSStnSeqProOutput.i8ProTankBtmUsAkHz := 0;
DSStnSeqProOutput.i9ProTankBtmUsBkHz := 0;
DSStnSeqProOutput.i10ProTankBtmUsCkHz := 0;
DSStnSeqProOutput.i11ProTankSideUsAkHz := 0;
DSStnSeqProOutput.i12ProTankSideUsBkHz := 0;
DSStnSeqProOutput.i13ProTankBlowerHz := 0;

DSStnSeqProOutput.r14ProTankChangeTempDegC := 0;
DSStnSeqProOutput.r15SubTankChangeTempDegC := 0;
DSStnSeqProOutput.i16SubTankPumpLPM := 0;
DSStnSeqProOutput.i17SubTankPumpHz := 0;

DSStnSeqProOutput.i18SlowPullVelocity := 0;
DSStnSeqProOutput.i19SlowPullDelayTime := 0;



END_IF

(*


(*[][][][][][][][][][][][][][][][][][][][][][][][][][][][][][][][][][][][][][][][][][][][][][][][][][][][][][][][][][][][][][][][][][][][][][][][]-Original FB StnSeqProcess Backup-[][][][][][][][][][][][][][][][][][][][][][][][][][][][][][][][][][][][][][][][][][][][][][][][][][][][][][][][][][][][][][][][][][][][][][][][]*)

(*[][][][][][][][][][][][][][][][][][]-Generate Current Process Time-[][][][][][][][][][][][][][][][][][]*)
tProcess1secClockPulse(IN:=bProcessInProgressFlag AND NOT tProcess1secClockPulse.Q , PT:= T#1s, Q=> , ET=> );
retProcess1secClockPulse(CLK:=tProcess1secClockPulse.Q , Q=> );

IF bProcessInProgressFlag AND retProcess1secClockPulse.Q THEN
iCurrentProcessTime := iCurrentProcessTime+1;
END_IF


(*[][][][][][][][][][][][][][][][][][]-Complete Condition Process Time Handling-[][][][][][][][][][][][][][][][][][]*)

(*Generate CompleteCondition Process Time Elapse Value (Reverse Counting)*)
IF bProcessInProgressFlag AND StationfbCallStnSeqSubPro.BufferDsSubRecipeMemory.bComCon20EnProcessTimer AND iStnSeqProcessCaseNo = 3 THEN
iComConProcessTimeEV := StationfbCallStnSeqSubPro.BufferDsSubRecipeMemory.iComCon5ProcessTimer - iComConProcessTime;
ELSE
iComConProcessTimeEV := 0;
END_IF


(*Start Complete Condition Timer If Available*)
tStartProcess1secClockPulse(IN:=StationfbCallStnSeqSubPro.BufferDsSubRecipeMemory.bComCon20EnProcessTimer AND NOT tProcess1secClockPulse.Q AND iStnSeqProcessCaseNo = 3 , PT:=T#1s , Q=> , ET=> );
retStartProcess1secClockPulse(CLK:=tStartProcess1secClockPulse.Q , Q=> );

IF bProcessInProgressFlag AND tStartProcess1secClockPulse.Q THEN
iComConProcessTime := iComConProcessTime+1;
END_IF

IF iComConProcessTime >= StationfbCallStnSeqSubPro.BufferDsSubRecipeMemory.iComCon5ProcessTimer THEN
bStationProcessTimerComplete := TRUE;
ELSE
bStationProcessTimerComplete := FALSE;
END_IF


(*[][][][][][][][][][][][][][][][][][]-Generate Above/Below-Start Condition-[][][][][][][][][][][][][][][][][][]*)

IF DsStnSeqProInput.iVacuumLevelPV < StationfbCallStnSeqSubPro.BufferDsSubRecipeMemory.iStCon1TargetVacuumLevel THEN
bStCon11BelowTargetVacuumLevel := TRUE;
ELSE
bStCon11BelowTargetVacuumLevel := FALSE;
END_IF

IF DsStnSeqProInput.iVacuumLevelPV >= StationfbCallStnSeqSubPro.BufferDsSubRecipeMemory.iStCon1TargetVacuumLevel THEN
bStCon12AboveTargetVacuumLevel := TRUE;
ELSE
bStCon12AboveTargetVacuumLevel := FALSE;
END_IF

IF DsStnSeqProInput.iPressureLevelPV < StationfbCallStnSeqSubPro.BufferDsSubRecipeMemory.iStCon2TargetPressureLevel THEN
bStCon13BelowTargetPressureLevel := TRUE;
ELSE
bStCon13BelowTargetPressureLevel := FALSE;
END_IF

IF DsStnSeqProInput.iPressureLevelPV >= StationfbCallStnSeqSubPro.BufferDsSubRecipeMemory.iStCon2TargetPressureLevel THEN
bStCon14AboveTargetPressureLevel := TRUE;
ELSE
bStCon14AboveTargetPressureLevel := FALSE;
END_IF

IF DsStnSeqProInput.iProTankTempLevelPV < StationfbCallStnSeqSubPro.BufferDsSubRecipeMemory.iStCon3TargetProTankTempLevel THEN
bStCon15BelowTargetProTankTempLevel := TRUE;
ELSE
bStCon15BelowTargetProTankTempLevel := FALSE;
END_IF

IF DsStnSeqProInput.iProTankTempLevelPV >= StationfbCallStnSeqSubPro.BufferDsSubRecipeMemory.iStCon3TargetProTankTempLevel THEN
bStCon16AboveTargetProTankTempLevel := TRUE;
ELSE
bStCon16AboveTargetProTankTempLevel := FALSE;
END_IF

IF DsStnSeqProInput.iSubTankTempLevelPV < StationfbCallStnSeqSubPro.BufferDsSubRecipeMemory.iStCon4TargetSubTankTempLevel THEN
bStCon15BelowTargetProTankTempLevel := TRUE;
ELSE
bStCon15BelowTargetProTankTempLevel := FALSE;
END_IF

IF DsStnSeqProInput.iSubTankTempLevelPV >= StationfbCallStnSeqSubPro.BufferDsSubRecipeMemory.iStCon4TargetSubTankTempLevel THEN
bStCon16AboveTargetProTankTempLevel := TRUE;
ELSE
bStCon16AboveTargetProTankTempLevel := FALSE;
END_IF


(*[][][][][][][][][][][][][][][][][][]-Generate Above/Below-Complete Condition-[][][][][][][][][][][][][][][][][][]*)

IF DsStnSeqProInput.iVacuumLevelPV < StationfbCallStnSeqSubPro.BufferDsSubRecipeMemory.iComCon1TargetVacuumLevel THEN
bComCon11BelowTargetVacuumLevel := TRUE;
ELSE
bComCon11BelowTargetVacuumLevel := FALSE;
END_IF

IF DsStnSeqProInput.iVacuumLevelPV >= StationfbCallStnSeqSubPro.BufferDsSubRecipeMemory.iComCon1TargetVacuumLevel THEN
bComCon12AboveTargetVacuumLevel := TRUE;
ELSE
bComCon12AboveTargetVacuumLevel := FALSE;
END_IF

IF DsStnSeqProInput.iPressureLevelPV < StationfbCallStnSeqSubPro.BufferDsSubRecipeMemory.iComCon2TargetPressureLevel THEN
bComCon13BelowTargetPressureLevel := TRUE;
ELSE
bComCon13BelowTargetPressureLevel := FALSE;
END_IF

IF DsStnSeqProInput.iPressureLevelPV >= StationfbCallStnSeqSubPro.BufferDsSubRecipeMemory.iComCon2TargetPressureLevel THEN
bComCon14AboveTargetPressureLevel := TRUE;
ELSE
bComCon14AboveTargetPressureLevel := FALSE;
END_IF

IF DsStnSeqProInput.iProTankTempLevelPV < StationfbCallStnSeqSubPro.BufferDsSubRecipeMemory.iComCon3TargetProTankTempLevel THEN
bComCon15BelowTargetProTankTempLevel := TRUE;
ELSE
bComCon15BelowTargetProTankTempLevel := FALSE;
END_IF

IF DsStnSeqProInput.iProTankTempLevelPV >= StationfbCallStnSeqSubPro.BufferDsSubRecipeMemory.iComCon3TargetProTankTempLevel THEN
bComCon16AboveTargetProTankTempLevel := TRUE;
ELSE
bComCon16AboveTargetProTankTempLevel := FALSE;
END_IF

IF DsStnSeqProInput.iSubTankTempLevelPV < StationfbCallStnSeqSubPro.BufferDsSubRecipeMemory.iComCon4TargetSubTankTempLevel THEN
bComCon17BelowTargetSubTankTempLevel := TRUE;
ELSE
bComCon17BelowTargetSubTankTempLevel := FALSE;
END_IF

IF DsStnSeqProInput.iSubTankTempLevelPV >= StationfbCallStnSeqSubPro.BufferDsSubRecipeMemory.iComCon4TargetSubTankTempLevel THEN
bComCon18AboveTargetSubTankTempLevel := TRUE;
ELSE
bComCon18AboveTargetSubTankTempLevel := FALSE;
END_IF

(*[][][][][][][][][][][][][][][][][][]-General-[][][][][][][][][][][][][][][][][][]*)
rebProcessHalt(CLK:=bProcessHalt , Q=> );

febProcessHalt(CLK:=bProcessHalt , Q=> );

IF rebProcessHalt.Q AND bProcessInProgressFlag THEN
bProcessInProgressFlag := FALSE;
bProcessHaltFlag := TRUE;
END_IF

IF febProcessHalt.Q AND bProcessHaltFlag THEN
bProcessInProgressFlag := TRUE;
bProcessHaltFlag := FALSE;
END_IF



IF bProcessReset OR NOT DsBasketInfo.bAvailibility THEN
bProcessInProgressFlag := FALSE;
bCallStnSeqRecipeErr := FALSE;
bInvalidProcessStepErr := FALSE;
bCallStnSeqSubProEn := FALSE;
bProcessCompleted := FALSE;
bProcessHaltFlag := FALSE;

iStnSeqProcessCaseNo := 0;
iCurrentProcessStep := 0;
iCurrentProcessTime := 0;
iComConProcessTime := 0;
ClearFL := 1;

	FOR ClearFL := 1 TO 10 DO
		ARiCurrentCycle[ClearFL] := 0;
	END_FOR

END_IF




rebProcessStart(CLK:=bProcessStart , Q=> );

IF rebProcessStart.Q THEN
iStnSeqProcessCaseNo := 1;
iCurrentProcessStep := 1;
ARiCurrentCycle[iCurrentProcessStep] := 1;
bProcessInProgressFlag := TRUE;
END_IF


(*[][][][][][][][][][][][][][][][][][]-FB Declaration-[][][][][][][][][][][][][][][][][][]*)

StationfbCallStnSeqSubPro(
	bCallSt:= bCallStnSeqSubProEn ,
	iCurrentProcessStep:=iCurrentProcessStep ,
	DSStnSeqRepCall:=DsStnSeqRepCall ,
	DSStnSeqSubCall:=DsStnSubRepCall ,
	DSBasketInfo:=DsBasketInfo ,
	bCallCompleted=>bTempCallCompleted ,
	bInvalidProcessStepErrHold=>bTempInvalidProcessStepErr ,
	bInvalidProcessStepErrPulse=>bTempInvalidProcessStepErrPls,
	bCallStnSeqRecipeErr=> bTempCallStnSeqRecipeErr,
	bCallStnSubRecipeErr=> bTempCallStnSubRecipeErr,
	BuffersSubDescription=> sTempsSubDescription,
	BufferDsSubRecipeMemory=> DsTempSubRecipeMemory,
	iSeqStep=> iTempSeqStep);


(*[][][][][][][][][][][][][][][][][][]-Stop Output when Process is Stop/Complete/Halt-[][][][][][][][][][][][][][][][][][]*)

IF NOT bProcessInProgressFlag THEN
DSStnSeqProOutput.b1ProTankPump := FALSE;
DSStnSeqProOutput.b2ProTankHeater := FALSE;
DSStnSeqProOutput.b3ProTankBottomUltrasonicA := FALSE;
DSStnSeqProOutput.b4ProTankBottomUltrasonicB := FALSE;
DSStnSeqProOutput.b5ProTankBottomUltrasonicC := FALSE;
DSStnSeqProOutput.b6ProTankSideUltrasonicA := FALSE;
DSStnSeqProOutput.b7ProTankSideUltrasonicB := FALSE;
DSStnSeqProOutput.b8SubTankPump := FALSE;
DSStnSeqProOutput.b9SubTankHeater := FALSE;
DSStnSeqProOutput.b10Blower := FALSE;
DSStnSeqProOutput.b11VacuumPump := FALSE;
DSStnSeqProOutput.b12Instrument1 := FALSE;
DSStnSeqProOutput.b13Instrument2 := FALSE;
DSStnSeqProOutput.b14Instrument3 := FALSE;
DSStnSeqProOutput.b15Instrument4 := FALSE;

DSStnSeqProOutput.b1ActValve1 := FALSE;
DSStnSeqProOutput.b2ActValve2 := FALSE;
DSStnSeqProOutput.b3ActValve3 := FALSE;
DSStnSeqProOutput.b4ActValve4 := FALSE;
DSStnSeqProOutput.b5ActValve5 := FALSE;
DSStnSeqProOutput.b6ActValve6 := FALSE;
DSStnSeqProOutput.b7ActValve7 := FALSE;
DSStnSeqProOutput.b8ActValve8 := FALSE;
DSStnSeqProOutput.b9ActValve9 := FALSE;
DSStnSeqProOutput.b10ActValve10 := FALSE;
DSStnSeqProOutput.b11ActValve11 := FALSE;
DSStnSeqProOutput.b12ActValve12 := FALSE;
DSStnSeqProOutput.b13ActValve13 := FALSE;
DSStnSeqProOutput.b14ActValve14 := FALSE;
DSStnSeqProOutput.b15ActValve15 := FALSE;

DSStnSeqProOutput.i1ProTankPumpLPM := 0;
DSStnSeqProOutput.i2ProTankPumpHz := 0;
DSStnSeqProOutput.i3ProTankBtmUsAPwrPercent := 0;
DSStnSeqProOutput.i4ProTankBtmUsBPwrPercent := 0;
DSStnSeqProOutput.i5ProTankBtmUsCPwrPercent := 0;
DSStnSeqProOutput.i6ProTankSideUsAPwrPercent := 0;
DSStnSeqProOutput.i7ProTankSideUsBPwrPercent := 0;
DSStnSeqProOutput.i8ProTankBtmUsAkHz := 0;
DSStnSeqProOutput.i9ProTankBtmUsBkHz := 0;
DSStnSeqProOutput.i10ProTankBtmUsCkHz := 0;
DSStnSeqProOutput.i11ProTankSideUsAkHz := 0;
DSStnSeqProOutput.i12ProTankSideUsBkHz := 0;
DSStnSeqProOutput.i13ProTankBlowerHz := 0;
END_IF

(*[][][][][][][][][][][][][][][][][][]-Main-Case/Step Programming-[][][][][][][][][][][][][][][][][][]*)

rebStnSeqSubCallCompleted(CLK:=StationfbCallStnSeqSubPro.bCallCompleted , Q=> );
rebCallStnSeqRecipeErr(CLK:=StationfbCallStnSeqSubPro.bCallStnSeqRecipeErr , Q=> );
rebInvalidProcessStepErr(CLK:=StationfbCallStnSeqSubPro.bInvalidProcessStepErrPulse , Q=> );
rebCallStnSubRecipeErr(CLK:=StationfbCallStnSeqSubPro.bCallStnSubRecipeErr , Q=> );


CASE iStnSeqProcessCaseNo OF

0:;

1: (*Pull Data from fbCallStnSeqSubPro*)
bCallStnSeqSubProEn:= TRUE;

IF rebStnSeqSubCallCompleted.Q THEN
bCallStnSeqSubProEn := FALSE;
bStartConditionPassed := FALSE;
bCompleteConditionPassed := FALSE;
iStnSeqProcessCaseNo := 2;
END_IF

IF rebCallStnSeqRecipeErr.Q THEN
bCallStnSeqSubProEn := FALSE;
bStartConditionPassed := FALSE;
bCompleteConditionPassed := FALSE;
iStnSeqProcessCaseNo := 90;
END_IF

IF rebInvalidProcessStepErr.Q THEN
bCallStnSeqSubProEn := FALSE;
bStartConditionPassed := FALSE;
bCompleteConditionPassed := FALSE;
iStnSeqProcessCaseNo := 91;
END_IF

IF rebCallStnSubRecipeErr.Q THEN
bCallStnSeqSubProEn := FALSE;
bStartConditionPassed := FALSE;
bCompleteConditionPassed := FALSE;
iStnSeqProcessCaseNo := 92;
END_IF

2: (*Start Condition Validation*)
IF bProcessInProgressFlag AND (
(StationfbCallStnSeqSubPro.BufferDsSubRecipeMemory.bStCon1EnLowLiquidLevel AND NOT DsStnSeqProInput.bLowLiquidLevel_NC) OR
(StationfbCallStnSeqSubPro.BufferDsSubRecipeMemory.bStCon2EnRegLiquidLevel AND DsStnSeqProInput.bRegLiquidLevel_NO) OR
(StationfbCallStnSeqSubPro.BufferDsSubRecipeMemory.bStCon3EnLowVacuumLevel AND DsStnSeqProInput.bLowVacuumLevel_NO) OR
(StationfbCallStnSeqSubPro.BufferDsSubRecipeMemory.bStCon4EnRegVacuumLevel AND DsStnSeqProInput.bRegVacuumLevel_NO) OR
(StationfbCallStnSeqSubPro.BufferDsSubRecipeMemory.bStCon5EnLowPressureLevel AND DsStnSeqProInput.bLowPressureLevel_NO) OR
(StationfbCallStnSeqSubPro.BufferDsSubRecipeMemory.bStCon6EnRegPressureLevel AND DsStnSeqProInput.bRegPressureLevel_NO) OR
(StationfbCallStnSeqSubPro.BufferDsSubRecipeMemory.bStCon7EnBelowTargetVacuumLevel AND bStCon11BelowTargetVacuumLevel) OR
(StationfbCallStnSeqSubPro.BufferDsSubRecipeMemory.bStCon8EnAboveTargetVacuumLevel AND bStCon12AboveTargetVacuumLevel) OR
(StationfbCallStnSeqSubPro.BufferDsSubRecipeMemory.bStCon9EnBelowTargetPressureLevel AND bStCon13BelowTargetPressureLevel) OR
(StationfbCallStnSeqSubPro.BufferDsSubRecipeMemory.bStCon10EnAboveTargetPressureLevel AND bStCon14AboveTargetPressureLevel) OR
(StationfbCallStnSeqSubPro.BufferDsSubRecipeMemory.bStCon11EnBelowTargetProTankTempLevel AND bStCon15BelowTargetProTankTempLevel) OR
(StationfbCallStnSeqSubPro.BufferDsSubRecipeMemory.bStCon12EnAboveTargetProTankTempLevel AND bStCon16AboveTargetProTankTempLevel) OR
(StationfbCallStnSeqSubPro.BufferDsSubRecipeMemory.bStCon13EnBelowTargetSubTankTempLevel AND bStCon17BelowTargetSubTankTempLevel) OR
(StationfbCallStnSeqSubPro.BufferDsSubRecipeMemory.bStCon14EnAboveTargetSubTankTempLevel AND bStCon18AboveTargetSubTankTempLevel) OR
(StationfbCallStnSeqSubPro.BufferDsSubRecipeMemory.bStCon15ExternalActivation AND DsStnSeqProInput.bExternalActivation_NO) OR

(NOT StationfbCallStnSeqSubPro.BufferDsSubRecipeMemory.bStCon1EnLowLiquidLevel
AND NOT StationfbCallStnSeqSubPro.BufferDsSubRecipeMemory.bStCon2EnRegLiquidLevel
AND NOT StationfbCallStnSeqSubPro.BufferDsSubRecipeMemory.bStCon3EnLowVacuumLevel
AND NOT StationfbCallStnSeqSubPro.BufferDsSubRecipeMemory.bStCon4EnRegVacuumLevel
AND NOT StationfbCallStnSeqSubPro.BufferDsSubRecipeMemory.bStCon5EnLowPressureLevel
AND NOT StationfbCallStnSeqSubPro.BufferDsSubRecipeMemory.bStCon6EnRegPressureLevel
AND NOT StationfbCallStnSeqSubPro.BufferDsSubRecipeMemory.bStCon7EnBelowTargetVacuumLevel
AND NOT StationfbCallStnSeqSubPro.BufferDsSubRecipeMemory.bStCon8EnAboveTargetVacuumLevel
AND NOT StationfbCallStnSeqSubPro.BufferDsSubRecipeMemory.bStCon9EnBelowTargetPressureLevel
AND NOT StationfbCallStnSeqSubPro.BufferDsSubRecipeMemory.bStCon10EnAboveTargetPressureLevel
AND NOT StationfbCallStnSeqSubPro.BufferDsSubRecipeMemory.bStCon11EnBelowTargetProTankTempLevel
AND NOT StationfbCallStnSeqSubPro.BufferDsSubRecipeMemory.bStCon12EnAboveTargetProTankTempLevel
AND NOT StationfbCallStnSeqSubPro.BufferDsSubRecipeMemory.bStCon13EnBelowTargetSubTankTempLevel
AND NOT StationfbCallStnSeqSubPro.BufferDsSubRecipeMemory.bStCon14EnAboveTargetSubTankTempLevel
AND NOT StationfbCallStnSeqSubPro.BufferDsSubRecipeMemory.bStCon15ExternalActivation) )THEN

bStartConditionPassed := TRUE;
iStnSeqProcessCaseNo := 3;
END_IF

3: (* Process Start Progress and Waiting Validate Complete Condition*)



(*Complete Condition Validation*)s
IF bProcessInProgressFlag AND (
(StationfbCallStnSeqSubPro.BufferDsSubRecipeMemory.bComCon1EnProLowLiquidLevel AND NOT DsStnSeqProInput.bProLowLiquidLevel_NC) OR
(StationfbCallStnSeqSubPro.BufferDsSubRecipeMemory.bComCon2EnProRegLiquidLevel AND DsStnSeqProInput.bProRegLiquidLevel_NO) OR
(StationfbCallStnSeqSubPro.BufferDsSubRecipeMemory.bComCon3EnProHighLiquidLevel AND DsStnSeqProInput.bProHighLiquidLevel_NO) OR
(StationfbCallStnSeqSubPro.BufferDsSubRecipeMemory.bComCon4EnSubLowLiquidLevel AND DsStnSeqProInput.bSubLowLiquidLevel_NC) OR
(StationfbCallStnSeqSubPro.BufferDsSubRecipeMemory.bComCon5EnSubRegLiquidLevel AND DsStnSeqProInput.bSubRegLiquidLevel_NO) OR
(StationfbCallStnSeqSubPro.BufferDsSubRecipeMemory.bComCon6EnSubHighLiquidLevel AND DsStnSeqProInput.bSubHighLiquidLevel_NO) OR

(StationfbCallStnSeqSubPro.BufferDsSubRecipeMemory.bComCon7EnLowVacuumLevel AND DsStnSeqProInput.bLowVacuumLevel_NO) OR
(StationfbCallStnSeqSubPro.BufferDsSubRecipeMemory.bComCon8EnRegVacuumLevel AND DsStnSeqProInput.bRegVacuumLevel_NO) OR
(StationfbCallStnSeqSubPro.BufferDsSubRecipeMemory.bComCon9EnLowPressureLevel AND DsStnSeqProInput.bLowPressureLevel_NO) OR
(StationfbCallStnSeqSubPro.BufferDsSubRecipeMemory.bComCon10EnRegPressureLevel AND DsStnSeqProInput.bRegPressureLevel_NO) OR
(StationfbCallStnSeqSubPro.BufferDsSubRecipeMemory.bComCon11EnBelowTargetVacuumLevel AND bComCon11BelowTargetVacuumLevel) OR
(StationfbCallStnSeqSubPro.BufferDsSubRecipeMemory.bComCon12EnAboveTargetVacuumLevel AND bComCon12AboveTargetVacuumLevel) OR
(StationfbCallStnSeqSubPro.BufferDsSubRecipeMemory.bComCon13EnBelowTargetPressureLevel AND bComCon13BelowTargetPressureLevel) OR
(StationfbCallStnSeqSubPro.BufferDsSubRecipeMemory.bComCon14EnAboveTargetPressureLevel AND bComCon14AboveTargetPressureLevel) OR
(StationfbCallStnSeqSubPro.BufferDsSubRecipeMemory.bComCon15EnBelowTargetProTankTempLevel AND bComCon15BelowTargetProTankTempLevel) OR
(StationfbCallStnSeqSubPro.BufferDsSubRecipeMemory.bComCon16EnAboveTargetProTankTempLevel AND bComCon16AboveTargetProTankTempLevel) OR
(StationfbCallStnSeqSubPro.BufferDsSubRecipeMemory.bComCon17EnBelowTargetSubTankTempLevel AND bComCon17BelowTargetSubTankTempLevel) OR
(StationfbCallStnSeqSubPro.BufferDsSubRecipeMemory.bComCon18EnAboveTargetSubTankTempLevel AND bComCon18AboveTargetSubTankTempLevel) OR
(StationfbCallStnSeqSubPro.BufferDsSubRecipeMemory.bComCon20EnProcessTimer AND bStationProcessTimerComplete) OR

(NOT StationfbCallStnSeqSubPro.BufferDsSubRecipeMemory.bComCon1EnProLowLiquidLevel
AND NOT StationfbCallStnSeqSubPro.BufferDsSubRecipeMemory.bComCon2EnProRegLiquidLevel
AND NOT StationfbCallStnSeqSubPro.BufferDsSubRecipeMemory.bComCon3EnProHighLiquidLevel
AND NOT StationfbCallStnSeqSubPro.BufferDsSubRecipeMemory.bComCon4EnSubLowLiquidLevel
AND NOT StationfbCallStnSeqSubPro.BufferDsSubRecipeMemory.bComCon5EnSubRegLiquidLevel
AND NOT StationfbCallStnSeqSubPro.BufferDsSubRecipeMemory.bComCon6EnSubHighLiquidLevel
AND NOT StationfbCallStnSeqSubPro.BufferDsSubRecipeMemory.bComCon7EnLowVacuumLevel
AND NOT StationfbCallStnSeqSubPro.BufferDsSubRecipeMemory.bComCon8EnRegVacuumLevel
AND NOT StationfbCallStnSeqSubPro.BufferDsSubRecipeMemory.bComCon9EnLowPressureLevel
AND NOT StationfbCallStnSeqSubPro.BufferDsSubRecipeMemory.bComCon10EnRegPressureLevel
AND NOT StationfbCallStnSeqSubPro.BufferDsSubRecipeMemory.bComCon11EnBelowTargetVacuumLevel
AND NOT StationfbCallStnSeqSubPro.BufferDsSubRecipeMemory.bComCon12EnAboveTargetVacuumLevel
AND NOT StationfbCallStnSeqSubPro.BufferDsSubRecipeMemory.bComCon13EnBelowTargetPressureLevel
AND NOT StationfbCallStnSeqSubPro.BufferDsSubRecipeMemory.bComCon14EnAboveTargetPressureLevel
AND NOT StationfbCallStnSeqSubPro.BufferDsSubRecipeMemory.bComCon15EnBelowTargetProTankTempLevel
AND NOT StationfbCallStnSeqSubPro.BufferDsSubRecipeMemory.bComCon16EnAboveTargetProTankTempLevel
AND NOT StationfbCallStnSeqSubPro.BufferDsSubRecipeMemory.bComCon17EnBelowTargetSubTankTempLevel
AND NOT StationfbCallStnSeqSubPro.BufferDsSubRecipeMemory.bComCon18EnAboveTargetSubTankTempLevel
AND NOT StationfbCallStnSeqSubPro.BufferDsSubRecipeMemory.bComCon20EnProcessTimer) )THEN

bCompleteConditionPassed := TRUE;
iStnSeqProcessCaseNo := 4;
END_IF


(*Trigger Output*)

IF bProcessInProgressFlag THEN
DSStnSeqProOutput.b1ProTankPump := StationfbCallStnSeqSubPro.BufferDsSubRecipeMemory.bOut1EnProTankPump;
DSStnSeqProOutput.b2ProTankHeater := StationfbCallStnSeqSubPro.BufferDsSubRecipeMemory.bOut2EnProTankHeater;
DSStnSeqProOutput.b3ProTankBottomUltrasonicA := StationfbCallStnSeqSubPro.BufferDsSubRecipeMemory.bOut3EnProTankBottomUltrasonicA;
DSStnSeqProOutput.b4ProTankBottomUltrasonicB := StationfbCallStnSeqSubPro.BufferDsSubRecipeMemory.bOut4EnProTankBottomUltrasonicB;
DSStnSeqProOutput.b5ProTankBottomUltrasonicC := StationfbCallStnSeqSubPro.BufferDsSubRecipeMemory.bOut5EnProTankBottomUltrasonicC;
DSStnSeqProOutput.b6ProTankSideUltrasonicA := StationfbCallStnSeqSubPro.BufferDsSubRecipeMemory.bOut6EnProTankSideUltrasonicA;
DSStnSeqProOutput.b7ProTankSideUltrasonicB := StationfbCallStnSeqSubPro.BufferDsSubRecipeMemory.bOut7EnProTankSideUltrasonicB;
DSStnSeqProOutput.b8SubTankPump := StationfbCallStnSeqSubPro.BufferDsSubRecipeMemory.bOut8EnSubTankPump;
DSStnSeqProOutput.b9SubTankHeater := StationfbCallStnSeqSubPro.BufferDsSubRecipeMemory.bOut9EnSubTankHeater;
DSStnSeqProOutput.b10Blower := StationfbCallStnSeqSubPro.BufferDsSubRecipeMemory.bOut10EnBlower;
DSStnSeqProOutput.b11VacuumPump := StationfbCallStnSeqSubPro.BufferDsSubRecipeMemory.bOut11EnVacuumPump;
DSStnSeqProOutput.b12Instrument1 := StationfbCallStnSeqSubPro.BufferDsSubRecipeMemory.bOut12EnInstrument1;
DSStnSeqProOutput.b13Instrument2 := StationfbCallStnSeqSubPro.BufferDsSubRecipeMemory.bOut13EnInstrument2;
DSStnSeqProOutput.b14Instrument3 := StationfbCallStnSeqSubPro.BufferDsSubRecipeMemory.bOut14EnInstrument3;
DSStnSeqProOutput.b15Instrument4 := StationfbCallStnSeqSubPro.BufferDsSubRecipeMemory.bOut15EnInstrument4;

DSStnSeqProOutput.b1ActValve1 := StationfbCallStnSeqSubPro.BufferDsSubRecipeMemory.bOut1ActValve1;
DSStnSeqProOutput.b2ActValve2 := StationfbCallStnSeqSubPro.BufferDsSubRecipeMemory.bOut2ActValve2;
DSStnSeqProOutput.b3ActValve3 := StationfbCallStnSeqSubPro.BufferDsSubRecipeMemory.bOut3ActValve3;
DSStnSeqProOutput.b4ActValve4 := StationfbCallStnSeqSubPro.BufferDsSubRecipeMemory.bOut4ActValve4;
DSStnSeqProOutput.b5ActValve5 := StationfbCallStnSeqSubPro.BufferDsSubRecipeMemory.bOut5ActValve5;
DSStnSeqProOutput.b6ActValve6 := StationfbCallStnSeqSubPro.BufferDsSubRecipeMemory.bOut6ActValve6;
DSStnSeqProOutput.b7ActValve7 := StationfbCallStnSeqSubPro.BufferDsSubRecipeMemory.bOut7ActValve7;
DSStnSeqProOutput.b8ActValve8 := StationfbCallStnSeqSubPro.BufferDsSubRecipeMemory.bOut8ActValve8;
DSStnSeqProOutput.b9ActValve9 := StationfbCallStnSeqSubPro.BufferDsSubRecipeMemory.bOut9ActValve9;
DSStnSeqProOutput.b10ActValve10 := StationfbCallStnSeqSubPro.BufferDsSubRecipeMemory.bOut10ActValve10;
DSStnSeqProOutput.b11ActValve11 := StationfbCallStnSeqSubPro.BufferDsSubRecipeMemory.bOut11ActValve11;
DSStnSeqProOutput.b12ActValve12 := StationfbCallStnSeqSubPro.BufferDsSubRecipeMemory.bOut12ActValve12;
DSStnSeqProOutput.b13ActValve13 := StationfbCallStnSeqSubPro.BufferDsSubRecipeMemory.bOut13ActValve13;
DSStnSeqProOutput.b14ActValve14 := StationfbCallStnSeqSubPro.BufferDsSubRecipeMemory.bOut14ActValve14;
DSStnSeqProOutput.b15ActValve15 := StationfbCallStnSeqSubPro.BufferDsSubRecipeMemory.bOut15ActValve15;

DSStnSeqProOutput.i1ProTankPumpLPM := StationfbCallStnSeqSubPro.BufferDsSubRecipeMemory.iOut1ProTankPumpLPM;
DSStnSeqProOutput.i2ProTankPumpHz := StationfbCallStnSeqSubPro.BufferDsSubRecipeMemory.iOut2ProTankPumpHz;
DSStnSeqProOutput.i3ProTankBtmUsAPwrPercent := StationfbCallStnSeqSubPro.BufferDsSubRecipeMemory.iOut3ProTankBtmUsAPwrPercent;
DSStnSeqProOutput.i4ProTankBtmUsBPwrPercent := StationfbCallStnSeqSubPro.BufferDsSubRecipeMemory.iOut4ProTankBtmUsBPwrPercent;
DSStnSeqProOutput.i5ProTankBtmUsCPwrPercent := StationfbCallStnSeqSubPro.BufferDsSubRecipeMemory.iOut5ProTankBtmUsCPwrPercent;
DSStnSeqProOutput.i6ProTankSideUsAPwrPercent := StationfbCallStnSeqSubPro.BufferDsSubRecipeMemory.iOut6ProTankSideUsAPwrPercent;
DSStnSeqProOutput.i7ProTankSideUsBPwrPercent := StationfbCallStnSeqSubPro.BufferDsSubRecipeMemory.iOut7ProTankSideUsBPwrPercent;
DSStnSeqProOutput.i8ProTankBtmUsAkHz := StationfbCallStnSeqSubPro.BufferDsSubRecipeMemory.iOut8ProTankBtmUsAkHz;
DSStnSeqProOutput.i9ProTankBtmUsBkHz := StationfbCallStnSeqSubPro.BufferDsSubRecipeMemory.iOut9ProTankBtmUsBkHz;
DSStnSeqProOutput.i10ProTankBtmUsCkHz := StationfbCallStnSeqSubPro.BufferDsSubRecipeMemory.iOut10ProTankBtmUsCkHz;
DSStnSeqProOutput.i11ProTankSideUsAkHz := StationfbCallStnSeqSubPro.BufferDsSubRecipeMemory.iOut11ProTankSideUsAkHz;
DSStnSeqProOutput.i12ProTankSideUsBkHz := StationfbCallStnSeqSubPro.BufferDsSubRecipeMemory.iOut12ProTankSideUsBkHz;
DSStnSeqProOutput.i13ProTankBlowerHz := StationfbCallStnSeqSubPro.BufferDsSubRecipeMemory.iOut13ProTankBlowerHz;
END_IF


4: (* Repeat Sequence *)

IF ARiCurrentCycle[iCurrentProcessStep] >= DsStnSeqRepCall.Call_DsStationSequenceRecipeMemory.AR10iCycle[iCurrentProcessStep] THEN

ARiCurrentCycle[iCurrentProcessStep] := 0;
iCurrentProcessStep := iCurrentProcessStep+1;
ARiCurrentCycle[iCurrentProcessStep] := ARiCurrentCycle[iCurrentProcessStep]  +1;
iStnSeqProcessCaseNo := 6;

ELSE
iCurrentProcessStepBuffer :=DsStnSeqRepCall.Call_DsStationSequenceRecipeMemory.AR10iRepeatFromStepNo[iCurrentProcessStep];
iStnSeqProcessCaseNo := 5;
END_IF

5: (*Move CurrentProcessStepBuffer to CurrentProcessStep*)
iCurrentProcessStep := iCurrentProcessStepBuffer;
ARiCurrentCycle[iCurrentProcessStep] := ARiCurrentCycle[iCurrentProcessStep]  +1;
iStnSeqProcessCaseNo := 6;

6: (* Trigger Repeat Process*)
bStartConditionPassed := FALSE;
bCompleteConditionPassed := FALSE;
iComConProcessTime := 0;
iStnSeqProcessCaseNo := 1;

90:(*Trigger Call Station Sequence Recipe Error*);
bCallStnSeqRecipeErr := TRUE;
bProcessInProgressFlag := FALSE;
iStnSeqProcessCaseNo := 97;

91:(*Trigger Invalid Process Step Error*)
bInvalidProcessStepErr := TRUE;
bProcessInProgressFlag := FALSE;
iStnSeqProcessCaseNo := 98;

92: (*Trigger Process Complete Flag*)
bProcessCompleted := TRUE;
bProcessInProgressFlag := FALSE;
iPreviousProcessTime := iCurrentProcessTime;
iCurrentProcessTime := 0;
iStnSeqProcessCaseNo := 99;


97:(*Stay if Call Station Sequence Recipe Error*)
;
98:(*Stay if Invalid Process Step Error*)
;
99:(*Stay if Process Completed*)
;

END_CASE

*)

END_FUNCTION_BLOCK

// ---- FBs/B_JKS_NewFB_V2/FBP-Memory_Sub/fbV2_StationSequenceRecipe.TcPOU
FUNCTION_BLOCK fbV2_StationSequenceRecipe

VAR_INPUT
	bSavePB  : BOOL;
	bLoadPB  : BOOL;
	bClearPB : BOOL;
	bCopyPB  : BOOL;
(*	iCopyFromSubRecipeNo : INT;*)
	iCopyToSubRecipeNo : INT;
	iStnID : INT;

END_VAR


VAR_IN_OUT PERSISTENT

	iStationSequenceRecipeNo							: INT; (* 10 sets of Station Sequence Recipe *)
	sStationSequenceRecipeDescription					 	: STRING(50); (* Description of Station Sequence Recipe - Naming*)
	DsInStationSequenceRecipeMemory 					: DSV2_StationSequenceRecipeMemory;
	ARDsSSERSourceMinMaxTime_Uni						: ARRAY [1..iStnQty] OF DSV2_SSERSourceMinMaxTime;
(*	AR10iStationSubProNo : ARRAY [0..10] OF INT; (* 10 units of SubProcessProgramNo / Steps *)
	AR10iCycle : ARRAY [0..10] OF INT; (* 10 units of Integer to Store the Cycle needed on the specified Steps. at least "1" *)
	AR10iRepeatFromStepNo : ARRAY [0..10] OF INT; (* 10 units of Integer to when Cycle repeat, it will repeat from Which Steps  *)
*)





	Call_iStationSequenceRecipe : INT;
	bCallPB: BOOL;
(*	bCallPBEnable : BOOL;*)
(*	ScrMapCall_iStationSequenceRecipe : INT;*)




END_VAR
VAR_OUTPUT
	bSaveInd : BOOL;
	bLoadInd : BOOL;
	bClearInd: BOOL;
	bCallCompleted : BOOL;
	bInvalidCallStationSequenceNoHold: BOOL;
	bInvalidCallStationSequenceNoPulse: BOOL;
(*	bInvalidScrMapCallStationSequenceNo : BOOL;*)
	Call_sSequenceRecipeDescription : STRING(50);
	Call_DsStationSequenceRecipeMemory : DSV2_StationSequenceRecipeMemory;

(*	Call_AR10iStationSubProNo : ARRAY [0..10] OF INT;
	Call_AR10iCycle : ARRAY [0..10] OF INT;
	Call_AR10iRepeatFromStepNo : ARRAY [0..10] OF INT;
*)
(*	ScrMapCall_sSequenceRecipeDescription : STRING(50);
	ScrMapCall_AR10iStationSubProNo : ARRAY [0..10] OF INT;
	ScrMapCall_AR10iCycle : ARRAY [0..10] OF INT;
	ScrMapCall_AR10iRepeatFromStepNo : ARRAY [0..10] OF INT;*)





END_VAR
VAR
	SaveIndHr: BOOL;
	LoadIndHr: BOOL;
	ClearIndHr: BOOL;

	SaveTimerDelay : TON;
	LoadTimerDelay : TON;
	ClearTimerDelay: TON;
	SelfCheckTimer: TON;
	bLoadEn: BOOL;
	SelfCheckloopSequenceRecipe: BOOL;
	PreviousNoSequenceRecipe: INT;

	LoadDF : R_TRIG;
	LoadENDF : R_TRIG;
	ClearDF : R_TRIG;
	SaveDF: R_TRIG;
	CallIntervalTimer: TON;
	CallIntervalDIFU: R_TRIG;

	bCallCompletedHR: BOOL;
	bCallCompletedHRRE: R_TRIG;
	CallCompletedTimer: TON;
	CallSelfCheckTimer : TON;
	CallSelfCheckloop : BOOL;

	CallSelfCheckRE: R_TRIG;
	CallStep: INT;
	CallSelfCheckHR: BOOL;
	bCallPBRE: R_TRIG;

	LoadFL: INT;
	SaveFL: INT;
	PreviousStationRequenceRecipeCallNo: INT;
	CallSFL: INT;
	febInvalidCallStationSequenceNo: F_TRIG;



	rebInvalidCallStationSequenceNo: R_TRIG;
	tInvalidCallStationSequenceNoPulseTimer: TON;
	CopyDF: R_TRIG;
	iMinMaxFL: INT;

	iCheckStepFL: INT;
	
	DSV2_StationSequenceRecipeMemory_Empty : DSV2_StationSequenceRecipeMemory;

END_VAR

VAR PERSISTENT

	ARDsStorageStationSequenceRecipeMemory : ARRAY [1..iStationSequenceRecipeArrayQty] OF DSV2_StationSequenceRecipeMemory;
	ARsStorageStationSequenceRecipeDescription: ARRAY [0..iStationSequenceRecipeArrayQty] OF STRING(50);


END_VAR

(*************Read MinMaxEffTime START***********************)

IF iStnID >= 1 AND iStnID <= iStnQty THEN

	iMinMaxFL := 1;
		FOR iMinMaxFL := 1 TO iStationSequenceRecipeArrayQty DO
			IF iMinMaxFL >= 1 AND iMinMaxFL <= iStationSequenceRecipeArrayQty THEN

				ARDsSSERSourceMinMaxTime_Uni[iStnID].ARiMinTime[iMinMaxFL] := ARDsStorageStationSequenceRecipeMemory[iMinMaxFL].iProcessMinTime;
				ARDsSSERSourceMinMaxTime_Uni[iStnID].ARiMaxTime[iMinMaxFL] := ARDsStorageStationSequenceRecipeMemory[iMinMaxFL].iProcessMaxTime;

			END_IF
		END_FOR

END_IF

(*************Read MinMaxEffTime END***********************)



IF iStationSequenceRecipeNo < 1 THEN
iStationSequenceRecipeNo := 1;
END_IF

IF iStationSequenceRecipeNo > iStationSequenceRecipeArrayQty THEN
iStationSequenceRecipeNo := iStationSequenceRecipeArrayQty;
END_IF

(*Add New*)
ARsStorageStationSequenceRecipeDescription[0] := '- - - End Step - - -';

(*Clear Indicator*)
IF bClearPB THEN
ClearIndHr := TRUE;
END_IF

ClearTimerDelay(IN:=ClearIndHr, PT := T#1S, Q=>, ET=>);
IF ClearTimerDelay.Q THEN
ClearIndHr := FALSE;
END_IF

IF ClearIndHr AND NOT ClearTimerDelay.Q THEN
bClearInd := TRUE;
ELSE
bClearInd := FALSE;
END_IF

(*Load and Save Indicator*)
IF bSavePB THEN
SaveIndHr := TRUE;
END_IF

SaveTimerDelay(IN:=SaveIndHr, PT := T#1s, Q=>, ET=>);
IF SaveTimerDelay.Q THEN
SaveIndHr := FALSE;
END_IF

IF SaveIndHr AND NOT SaveTimerDelay.Q THEN
bSaveInd := TRUE;
ELSE
bSaveInd := FALSE;
END_IF

IF bLoadPB THEN
LoadIndHr := TRUE;
END_IF

LoadTimerDelay(IN:=LoadIndHr, PT := T#1s, Q=>, ET=>);
IF loadtimerdelay.Q THEN
LoadIndHr := FALSE;
END_IF

IF loadIndHr AND NOT LoadTimerDelay.Q THEN
bLoadInd := TRUE;
ELSE
bLoadInd := FALSE;
END_IF

IF iStationSequenceRecipeNo <> PreviousNoSequenceRecipe THEN
bLoadEn := TRUE;
ELSE
bLoadEn := FALSE;
END_IF


(*
(* Add Min Time Control - for Vacuum Tank*)

IF DsInStationSequenceRecipeMemory.iProcessMinTime > 0 AND DsInStationSequenceRecipeMemory.iPreFixOverallProcessMinTime > 0 THEN
	IF (DsInStationSequenceRecipeMemory.iProcessMinTime / DsInStationSequenceRecipeMemory.iPreFixOverallProcessMinTime) > 0 THEN
		DsInStationSequenceRecipeMemory.iPreFixCalculatedCycle := (DsInStationSequenceRecipeMemory.iProcessMinTime / DsInStationSequenceRecipeMemory.iPreFixOverallProcessMinTime) ;
	ELSE
		DsInStationSequenceRecipeMemory.iPreFixCalculatedCycle := 1 ;
	END_IF
END_IF
(*
iCheckStepFL := 1;
IF iCheckStepFL > 0 AND iCheckStepFL < iStationSequenceRecipeArrayQty THEN
	FOR iCheckStepFL := 1 TO iStationSequenceRecipeArrayQty DO
		IF DsInStationSequenceRecipeMemory.AR10iStationSubProNo[iCheckStepFL] = DsInStationSequenceRecipeMemory.iPreFixOverwriteStep_Cycle THEN
*)			DsInStationSequenceRecipeMemory.AR10iCycle[DsInStationSequenceRecipeMemory.iPreFixOverwriteStep_Cycle] := DsInStationSequenceRecipeMemory.iPreFixCalculatedCycle;
(*		END_IF
	END_FOR
END_IF
*)
*)






(* Load Recipe *)

LoadDF(CLK:=bLoadPB,Q=>);
LoadENDF(CLK:=bLoadEn,Q=>);

IF LoadDF.Q OR LoadENDF.Q THEN

DsInStationSequenceRecipeMemory := ARDsStorageStationSequenceRecipeMemory[iStationSequenceRecipeNo];
sStationSequenceRecipeDescription := ARsStorageStationSequenceRecipeDescription[iStationSequenceRecipeNo];
PreviousNoSequenceRecipe := iStationSequenceRecipeNo  ;

END_IF


(* Save Recipe *)

SaveDF(CLK:=bSavePB,Q=>);

IF SaveDF.Q THEN

ARDsStorageStationSequenceRecipeMemory[iStationSequenceRecipeNo] := DsInStationSequenceRecipeMemory;
ARsStorageStationSequenceRecipeDescription[iStationSequenceRecipeNo] := sStationSequenceRecipeDescription;

END_IF


(*Copy Recipe*)

CopyDF(CLK:=bCopyPB,Q=>);

IF CopyDF.Q THEN

ARDsStorageStationSequenceRecipeMemory[iCopyToSubRecipeNo] := ARDsStorageStationSequenceRecipeMemory[iStationSequenceRecipeNo];
ARsStorageStationSequenceRecipeDescription[iCopyToSubRecipeNo] := ARsStorageStationSequenceRecipeDescription[iStationSequenceRecipeNo];

END_IF

(* Clear Recipe *)

ClearDF(CLK:=bClearPB,Q=>);

IF ClearDF.Q THEN

ARDsStorageStationSequenceRecipeMemory[iStationSequenceRecipeNo] 		:=DSV2_StationSequenceRecipeMemory_Empty;
ARsStorageStationSequenceRecipeDescription[iStationSequenceRecipeNo] 	:= '';

END_IF


(* Call Recipe *)
(* ---- Call Recipe Complete Flag ---*)

(*
CallCompletedTimer(IN:=bCallCompleted , PT:=t#0.5s , Q=> , ET=> );
*)
IF (*CallCompletedTimer.Q*) NOT bCallPB THEN
bCallCompleted := FALSE;
END_IF
(*
CallSelfCheckRE(CLK:=PreviousStationRequenceRecipeCallNo <> Call_iStationSequenceRecipe , Q=> );

IF CallSelfCheckRE.Q THEN
CallSelfCheckHR := TRUE;
END_IF
*)
bCallPBRE(CLK:=bCallPB , Q=> );

IF (Call_iStationSequenceRecipe <= 0 OR Call_iStationSequenceRecipe > iStationSequenceRecipeArrayQty) AND bCallPB THEN
bInvalidCallStationSequenceNoHold := TRUE;
ELSE
bInvalidCallStationSequenceNoHold := FALSE;
END_IF


rebInvalidCallStationSequenceNo(CLK:= bCallPB AND bInvalidCallStationSequenceNoHold  , Q=> );

IF rebInvalidCallStationSequenceNo.Q THEN
bInvalidCallStationSequenceNoPulse := TRUE;
END_IF

tInvalidCallStationSequenceNoPulseTimer(IN:=bInvalidCallStationSequenceNoPulse , PT:=t#0.5s , Q=> , ET=> );

IF tInvalidCallStationSequenceNoPulseTimer.Q OR NOT bCallPB THEN
bInvalidCallStationSequenceNoPulse := FALSE;
END_IF
(*
febInvalidCallStationSequenceNo(CLK:=bInvalidCallStationSequenceNoHold  , Q=> );
*)
IF bCallPBRE.Q AND NOT bInvalidCallStationSequenceNoHold (*OR febInvalidCallStationSequenceNo.Q*) THEN
bCallCompleted := FALSE;
CallStep:= 1;
END_IF


CASE CallStep OF

1:

Call_DsStationSequenceRecipeMemory := ARDsStorageStationSequenceRecipeMemory[Call_iStationSequenceRecipe];
Call_sSequenceRecipeDescription := ARsStorageStationSequenceRecipeDescription[Call_iStationSequenceRecipe];

(*IF NOT bCallPBEnable AND CallSelfCheckHR THEN
CallStep := 10;
ELSIF NOT bCallPBEnable AND NOT CallSelfCheckHR THEN
CallStep := 99;*)


(*IF bCallPBEnable THEN*)
CallStep := 11;


10:
bCallCompleted := TRUE;
CallSelfCheckHR := FALSE;
PreviousStationRequenceRecipeCallNo := Call_iStationSequenceRecipe;
CallStep := 99;

11:

(*IF bCallPBEnable AND bCallPB THEN*)
bCallCompleted := TRUE;
(*ELSE
bCallCompleted := FALSE;*)
CallStep := 99;



99:
(*
bCallCompleted := FALSE;
*)
;
END_CASE

END_FUNCTION_BLOCK

// ---- FBs/B_JKS_NewFB/FBP-Memory_Sub/fbStationSubRecipe.TcPOU
FUNCTION_BLOCK fbStationSubRecipe

VAR_INPUT
	bSavePB : BOOL;
	bLoadPB : BOOL;
	bClearPB: BOOL;
	bCopyPB : BOOL;
(*	iCopyFromSubRecipeNo : INT;*)
	iCopyToSubRecipeNo : INT;
	DsStnSeqProInput 				: DS_StnSeqProInput;						(* Input - PV of Instrument (Temperature, pressure, vacuum and etc), Signal of Sensor to allowed program under the current station status.*)

END_VAR


VAR_IN_OUT PERSISTENT
	iSubRecipeNo : INT; (* x sets of Sub Recipe *)
	sSubRecipeDescription : STRING(50); (* Description of Sub Recipe - Naming*)
	DsInSubRecipeMemory : DS_SubRecipeMemory;

	Call_iSubRecipe : INT;
	bCallPB: BOOL;
(*	bCallPBEnable : BOOL;*)



END_VAR
VAR_OUTPUT
	bSaveInd: BOOL;
	bLoadInd: BOOL;
	bClearInd: BOOL;
	bCallCompleted : BOOL;

	bInvalidCallSubRecipeNoHold: BOOL;
	bInvalidCallSubRecipeNoPulse: BOOL;


	Call_sSubDescription : STRING(50);
	Call_DsSubRecipeMemory : DS_SubRecipeMemory;


END_VAR
VAR
	SaveIndHr	: BOOL;
	LoadIndHr	: BOOL;
	ClearIndHr  : BOOL;

	SaveTimerDelay: TON;
	LoadTimerDelay: TON;
	ClearTimerDelay: TON;
	SelfCheckTimer: TON;
	bLoadEn: BOOL;
	SelfCheckloopSub: BOOL;
	SelfCheckloopMain: BOOL;
	PreviousNoMain: INT;
	PreviousNoSub: INT;

	LoadDF : R_TRIG;
	LoadENDF : R_TRIG;
	ClearDF : R_TRIG;
	SaveDF: R_TRIG;
	CallIntervalTimer: TON;
	CallIntervalDIFU: R_TRIG;
	CallMFL: INT;

	bCallCompletedHR: BOOL;
	bCallCompletedHRRE: R_TRIG;
	CallCompletedTimer: TON;
	CallSelfCheckTimer : TON;
	CallSelfCheckloop : BOOL;
	PreviousCallNo : INT;

	CallSelfCheckRE: R_TRIG;
	CallStep: INT;
	CallSelfCheckHR: BOOL;
	bCallPBRE: R_TRIG;

	febInvalidCallSubRecipeNo: F_TRIG;

	rebInvalidCallSubRecipeNo: R_TRIG;
	tInvalidCallStationSubNoPulseTimer: TON;
	CopyDF: R_TRIG;
	
	DsSubRecipeMemory_Empty 			   : DS_SubRecipeMemory; 
END_VAR

VAR PERSISTENT
	ARDsStorageSubRecipeMemory : ARRAY [1..IStationSubRecipeArrayQty] OF DS_SubRecipeMemory;

	ARsStorageSubDescription: ARRAY [0..IStationSubRecipeArrayQty] OF STRING(50);


END_VAR

IF iSubRecipeNo < 1 THEN
iSubRecipeNo := 1;
END_IF

IF iSubRecipeNo > IStationSubRecipeArrayQty THEN
iSubRecipeNo := IStationSubRecipeArrayQty;
END_IF



(*Add new*)
ARsStorageSubDescription[0] := '- - - End Step - - -';

(*Clear Indicator*)
IF bClearPB THEN
ClearIndHr := TRUE;
END_IF

ClearTimerDelay(IN:=ClearIndHr, PT := T#1S, Q=>, ET=>);
IF ClearTimerDelay.Q THEN
ClearIndHr := FALSE;
END_IF

IF ClearIndHr AND NOT ClearTimerDelay.Q THEN
bClearInd := TRUE;
ELSE
bClearInd := FALSE;
END_IF

(*Load and Save Indicator*)
IF bSavePB THEN
SaveIndHr := TRUE;
END_IF

SaveTimerDelay(IN:=SaveIndHr, PT := T#1s, Q=>, ET=>);
IF SaveTimerDelay.Q THEN
SaveIndHr := FALSE;
END_IF

IF SaveIndHr AND NOT SaveTimerDelay.Q THEN
bSaveInd := TRUE;
ELSE
bSaveInd := FALSE;
END_IF

IF bLoadPB THEN
LoadIndHr := TRUE;
END_IF

LoadTimerDelay(IN:=LoadIndHr, PT := T#1s, Q=>, ET=>);
IF loadtimerdelay.Q THEN
LoadIndHr := FALSE;
END_IF

IF loadIndHr AND NOT LoadTimerDelay.Q THEN
bLoadInd := TRUE;
ELSE
bLoadInd := FALSE;
END_IF


IF iSubRecipeNo <> PreviousNoSub THEN
bLoadEn := TRUE;
ELSE
bLoadEn := FALSE;
END_IF

(* Add for Slow Pull*)
IF DsInSubRecipeMemory.bOut12EnSlowPull THEN
	IF DsStnSeqProInput.iSlowPullUpPos > 0 AND DsStnSeqProInput.iSlowPullDownPos > 0 AND DsInSubRecipeMemory.iOut18SlowPullVelocity >0 THEN
			IF DsInSubRecipeMemory.iComCon5ProcessTimer <
			(((DsStnSeqProInput.iSlowPullUpPos-DsStnSeqProInput.iSlowPullDownPos) / (DsInSubRecipeMemory.iOut18SlowPullVelocity))+1)
			THEN
				DsInSubRecipeMemory.iComCon5ProcessTimer := (((DsStnSeqProInput.iSlowPullUpPos-DsStnSeqProInput.iSlowPullDownPos) / (DsInSubRecipeMemory.iOut18SlowPullVelocity))+1);
			END_IF

			DsInSubRecipeMemory.iOut19SlowPullDelayTime :=
			DsInSubRecipeMemory.iComCon5ProcessTimer -
			(((DsStnSeqProInput.iSlowPullUpPos-DsStnSeqProInput.iSlowPullDownPos) / (DsInSubRecipeMemory.iOut18SlowPullVelocity))+1) ;

	ELSE
	DsInSubRecipeMemory.iOut19SlowPullDelayTime :=0;

	END_IF
END_IF





(* Load Recipe *)

LoadDF(CLK:=bLoadPB,Q=>);
LoadENDF(CLK:=bLoadEn,Q=>);

IF LoadDF.Q OR LoadENDF.Q THEN

DsInSubRecipeMemory := ARDsStorageSubRecipeMemory[iSubRecipeNo];
sSubRecipeDescription := ARsStorageSubDescription[iSubRecipeNo];
PreviousNoSub := iSubRecipeNo;

END_IF


(* Save Recipe *)

SaveDF(CLK:=bSavePB,Q=>);

IF SaveDF.Q THEN

ARDsStorageSubRecipeMemory[iSubRecipeNo] := DsInSubRecipeMemory;
ARsStorageSubDescription[iSubRecipeNo] := sSubRecipeDescription;

END_IF

(*Copy Recipe*)

CopyDF(CLK:=bCopyPB,Q=>);

IF CopyDF.Q THEN

ARDsStorageSubRecipeMemory[iCopyToSubRecipeNo] := ARDsStorageSubRecipeMemory[iSubRecipeNo];
ARsStorageSubDescription[iCopyToSubRecipeNo] := ARsStorageSubDescription[iSubRecipeNo];

END_IF

ClearDF(CLK:=bClearPB,Q=>);

IF ClearDF.Q THEN

ARDsStorageSubRecipeMemory[iSubRecipeNo] 		:=DsSubRecipeMemory_Empty;
ARsStorageSubDescription[iSubRecipeNo] 			:= '';

END_IF



(* Call Recipe *)
(* ---- Call Recipe Complete Flag ---*)

(*
CallCompletedTimer(IN:=bCallCompleted , PT:=t#0.5s , Q=> , ET=> );
*)
IF (*CallCompletedTimer.Q*) NOT bCallPB THEN
bCallCompleted := FALSE;
END_IF
(*
CallSelfCheckRE(CLK:=PreviousCallNo <> Call_iSubRecipe , Q=> );

IF CallSelfCheckRE.Q THEN
CallSelfCheckHR := TRUE;
END_IF
*)
bCallPBRE(CLK:=bCallPB , Q=> );

IF (Call_iSubRecipe <=0 OR Call_iSubRecipe > IStationSubRecipeArrayQty) AND bCallPB THEN
bInvalidCallSubRecipeNoHold := TRUE;
ELSE
bInvalidCallSubRecipeNoHold := FALSE;
END_IF

rebInvalidCallSubRecipeNo(CLK:= bCallPB AND bInvalidCallSubRecipeNoHold, Q=> );

IF rebInvalidCallSubRecipeNo.Q THEN
bInvalidCallSubRecipeNoPulse := TRUE;
END_IF

tInvalidCallStationSubNoPulseTimer(IN:=bInvalidCallSubRecipeNoPulse , PT:=t#0.5s , Q=> , ET=> );

IF tInvalidCallStationSubNoPulseTimer.Q OR NOT bCallPB THEN
bInvalidCallSubRecipeNoPulse := FALSE;
END_IF

(*
febInvalidCallSubRecipeNo(CLK:=bInvalidCallSubRecipeNoHold , Q=> );
*)
IF (bCallPBRE.Q AND NOT bInvalidCallSubRecipeNoHold) (*OR febInvalidCallSubRecipeNo.Q*) THEN
bCallCompleted := FALSE;
CallStep:= 1;
END_IF
CASE CallStep OF

1:

Call_DsSubRecipeMemory := ARDsStorageSubRecipeMemory[Call_iSubRecipe];
Call_sSubDescription := ARsStorageSubDescription[Call_iSubRecipe];
(*
IF NOT bCallPBEnable AND CallSelfCheckHR THEN
CallStep := 10;
END_IF

IF bCallPBEnable THEN*)
CallStep := 11;
(*END_IF*)

10:
bCallCompleted := TRUE;
CallSelfCheckHR := FALSE;
PreviousCallNo := Call_iSubRecipe;
CallStep := 99;

11:
(*
IF bCallPBEnable AND bCallPB THEN*)
bCallCompleted := TRUE;
CallStep := 99;




99:;

END_CASE

END_FUNCTION_BLOCK

// ---- FBs/B_JKS_NewFB_V2/FBP-Memory_Sub/fbV2_CallStnSeqSubPro.TcPOU
FUNCTION_BLOCK fbV2_CallStnSeqSubPro
VAR_INPUT
	bCallSt: BOOL;
	iCurrentProcessStep: INT;
END_VAR
VAR_OUTPUT PERSISTENT
	bCallCompleted : BOOL;
	bInvalidProcessStepErrHold : BOOL;
	bInvalidProcessStepErrPulse: BOOL;
	bCallStnSeqRecipeErr : BOOL;
	bCallStnSubRecipeErr : BOOL;
	BuffersSubDescription : STRING(50);
	BufferDsSubRecipeMemory : DS_SubRecipeMemory;
(*	BufferAR30iInt : ARRAY [0..30] OF INT;
	BufferAR50bBool : ARRAY [0..50] OF BOOL;
	BufferAR5sString : ARRAY [0..5] OF STRING(50);
	BufferAR5lrLreal : ARRAY [0..5] OF LREAL;*)
	iSeqStep: INT;
END_VAR

VAR_IN_OUT PERSISTENT

	DSStnSeqRepCall: DSV2_fbStationSequenceRecipeCall;
	DSStnSeqSubCall: DS_fbStationSubRecipeCall;
	DSBasketInfo : DSV2_BasketInfo;


END_VAR

VAR PERSISTENT


END_VAR
VAR
	CallSelfCheckHR: BOOL;
	iPreviousProcessStep: INT;
	CallSelfCheckRE : R_TRIG;
	febInvalidProcessStep : F_TRIG;

	reCallCompleted: R_TRIG;
	CallCompletedTimer: TON;

	rebInvalidStnSeqRepCall: R_TRIG;
	rebInvalidStnSubRepCall: R_TRIG;
	rebCallSt: R_TRIG;
	tCallStnSeqRecipeErrTimer: TON;
	tCallStnSubRecipeErrTimer: TON;
	tInvalidProcessStepErrTimer: TON;
	rebInvalidProcessStep: R_TRIG;
	BufferDsSubRecipeMemoryEmpty : DS_SubRecipeMemory;
END_VAR

(*Reset fb*)
IF NOT bCallSt THEN
DSStnSeqRepCall.bCallPB := FALSE;
DSStnSeqSubCall.bCallPB := FALSE;
bCallCompleted := FALSE;
bCallStnSeqRecipeErr := FALSE;
bCallStnSubRecipeErr := FALSE;
iSeqStep := 0;
(*BuffersSubDescription := '' ;
BufferDsSubRecipeMemory := BufferDsSubRecipeMemoryEmpty;
*)
END_IF


(*Reset Err after 0.5Sec*)

tCallStnSeqRecipeErrTimer(IN:= bCallStnSeqRecipeErr , PT:=t#0.5s , Q=> , ET=> );

IF tCallStnSeqRecipeErrTimer.Q OR NOT bCallSt THEN
bCallStnSeqRecipeErr := FALSE;
END_IF


tCallStnSubRecipeErrTimer(IN:= bCallStnSubRecipeErr , PT:=t#0.5s , Q=> , ET=> );

IF tCallStnSubRecipeErrTimer.Q OR NOT bCallSt THEN
bCallStnSubRecipeErr := FALSE;
END_IF



(*Check if CurrentProcessStep changed, pull data from SSER and SSUR again*)

(*
CallSelfCheckRE(CLK:=iPreviousProcessStep <> iCurrentProcessStep , Q=> );

IF CallSelfCheckRE.Q THEN
CallSelfCheckHR := TRUE;
END_IF
*)
IF( iCurrentProcessStep <= 0 OR iCurrentProcessStep > iProductRecipeStepArrayQty) AND bCallSt THEN
bInvalidProcessStepErrHold := TRUE;
ELSE
bInvalidProcessStepErrHold := FALSE;
END_IF
(*
febInvalidProcessStep(CLK:=bInvalidProcessStepErrHold , Q=> );
*)
rebInvalidProcessStep(CLK:=bInvalidProcessStepErrHold AND bCallSt , Q=> );

IF rebInvalidProcessStep.Q THEN
bInvalidProcessStepErrPulse := TRUE;
END_IF


tInvalidProcessStepErrTimer(IN:= bInvalidProcessStepErrPulse , PT:=t#0.5s , Q=> , ET=> );

IF tInvalidProcessStepErrTimer.Q OR NOT bCallSt THEN
bInvalidProcessStepErrPulse := FALSE;
END_IF

(*Sequence Start*)
(*
IF NOT bSequenceSt THEN
iSeqStep := 0;
END_IF
*)
rebCallSt(CLK:=bCallSt , Q=> );
IF rebCallSt.Q (*OR (CallSelfCheckRE.Q*) AND NOT bInvalidProcessStepErrHold(*) OR febInvalidProcessStep.Q*) THEN
iSeqStep := 1;
(*BufferDsSubRecipeMemory.iComCon5ProcessTimer := -1 (* -1 is the reference if the calling have problem, it will shown -1 after call completed*);
*)
(*iCurrentProcessStep := 1;*)
END_IF

rebInvalidStnSeqRepCall(CLK:=DSStnSeqRepCall.bInvalidCallStationSequenceNoPulse , Q=> );
rebInvalidStnSubRepCall(CLK:=DSStnSeqSubCall.bInvalidCallSubRecipeNoPulse , Q=> );


CASE iSeqStep OF

0:;

1: (*Select Sequence Recipe By Refering Basket Information*)
bCallStnSeqRecipeErr := FALSE;
bCallStnSubRecipeErr := FALSE;

DSStnSeqRepCall.Call_iStationSequenceRecipe := DSBasketInfo.iStationSeqenceRecipeNo(*iProgramNo*);
DSStnSeqRepCall.bCallPB := TRUE;

IF DSStnSeqRepCall.bCallCompleted THEN
DSStnSeqRepCall.bCallPB := FALSE;

iSeqStep:=2;

END_IF

IF rebInvalidStnSeqRepCall.Q THEN
DSStnSeqRepCall.bCallPB := FALSE;

iSeqStep:=11;
END_IF



2: (*Select Sub Recipe By Refering Selected Sequence Recipe Number*)

DSStnSeqSubCall.Call_iSubRecipe := DSStnSeqRepCall.Call_DsStationSequenceRecipeMemory.AR10iStationSubProNo[iCurrentProcessStep];
DSStnSeqSubCall.bCallPB := TRUE;


IF DSStnSeqSubCall.bCallCompleted THEN
DSStnSeqSubCall.bCallPB := FALSE;

iSeqStep:=3;
END_IF

IF rebInvalidStnSubRepCall.Q THEN
DSStnSeqSubCall.bCallPB := FALSE;

iSeqStep:=12;
END_IF


3: (*Transfer Sub Recipe Detail to Buffer*)

	BuffersSubDescription := DSStnSeqSubCall.Call_sSubDescription ;
	BufferDsSubRecipeMemory := DSStnSeqSubCall.Call_DsSubRecipeMemory;

iSeqStep:=4;

4: (*Check if the calling value is ok*)
(*IF BufferDsSubRecipeMemory.iComCon5ProcessTimer <> -1 THEN*)
iPreviousProcessStep := iCurrentProcessStep;
bCallCompleted := TRUE;
CallSelfCheckHR := FALSE;
iSeqStep := 5;
(*END_IF*)
5:

CallCompletedTimer(IN:= bCallCompleted , PT:=t#0.5s , Q=> , ET=> );

IF CallCompletedTimer.Q THEN
bCallCompleted := FALSE;
END_IF


11:
iPreviousProcessStep := iCurrentProcessStep;
CallSelfCheckHR := FALSE;
bCallStnSeqRecipeErr := TRUE;
iSeqStep:=21;

12:
iPreviousProcessStep := iCurrentProcessStep;
bCallStnSubRecipeErr := TRUE;
CallSelfCheckHR := FALSE;
iSeqStep:=22;

21:;

22:;


END_CASE

END_FUNCTION_BLOCK

// ---- FBs/B_JKS_NewFB/FBP-Memory_Sub/fbCallStnSeqSubPro.TcPOU
FUNCTION_BLOCK fbCallStnSeqSubPro
VAR_INPUT
	bCallSt: BOOL;
	iCurrentProcessStep: INT;
END_VAR
VAR_OUTPUT PERSISTENT
	bCallCompleted : BOOL;
	bInvalidProcessStepErrHold : BOOL;
	bInvalidProcessStepErrPulse: BOOL;
	bCallStnSeqRecipeErr : BOOL;
	bCallStnSubRecipeErr : BOOL;
	BuffersSubDescription : STRING(50);
	BufferDsSubRecipeMemory : DS_SubRecipeMemory;
(*	BufferAR30iInt : ARRAY [0..30] OF INT;
	BufferAR50bBool : ARRAY [0..50] OF BOOL;
	BufferAR5sString : ARRAY [0..5] OF STRING(50);
	BufferAR5lrLreal : ARRAY [0..5] OF LREAL;*)
	iSeqStep: INT;
END_VAR

VAR_IN_OUT PERSISTENT

	DSStnSeqRepCall: DS_fbStationSequenceRecipeCall;
	DSStnSeqSubCall: DS_fbStationSubRecipeCall;
	DSBasketInfo : DS_BasketInfo;


END_VAR

VAR PERSISTENT


END_VAR
VAR
	CallSelfCheckHR: BOOL;
	iPreviousProcessStep: INT;
	CallSelfCheckRE : R_TRIG;
	febInvalidProcessStep : F_TRIG;

	reCallCompleted: R_TRIG;
	CallCompletedTimer: TON;

	rebInvalidStnSeqRepCall: R_TRIG;
	rebInvalidStnSubRepCall: R_TRIG;
	rebCallSt: R_TRIG;
	tCallStnSeqRecipeErrTimer: TON;
	tCallStnSubRecipeErrTimer: TON;
	tInvalidProcessStepErrTimer: TON;
	rebInvalidProcessStep: R_TRIG;
END_VAR

(*Reset fb*)
IF NOT bCallSt THEN
DSStnSeqRepCall.bCallPB := FALSE;
DSStnSeqSubCall.bCallPB := FALSE;
bCallCompleted := FALSE;
bCallStnSeqRecipeErr := FALSE;
bCallStnSubRecipeErr := FALSE;
iSeqStep := 0;

END_IF


(*Reset Err after 0.5Sec*)

tCallStnSeqRecipeErrTimer(IN:= bCallStnSeqRecipeErr , PT:=t#0.5s , Q=> , ET=> );

IF tCallStnSeqRecipeErrTimer.Q OR NOT bCallSt THEN
bCallStnSeqRecipeErr := FALSE;
END_IF


tCallStnSubRecipeErrTimer(IN:= bCallStnSubRecipeErr , PT:=t#0.5s , Q=> , ET=> );

IF tCallStnSubRecipeErrTimer.Q OR NOT bCallSt THEN
bCallStnSubRecipeErr := FALSE;
END_IF



(*Check if CurrentProcessStep changed, pull data from SSER and SSUR again*)

(*
CallSelfCheckRE(CLK:=iPreviousProcessStep <> iCurrentProcessStep , Q=> );

IF CallSelfCheckRE.Q THEN
CallSelfCheckHR := TRUE;
END_IF
*)
IF( iCurrentProcessStep <= 0 OR iCurrentProcessStep > iProductRecipeStepArrayQty) AND bCallSt THEN
bInvalidProcessStepErrHold := TRUE;
ELSE
bInvalidProcessStepErrHold := FALSE;
END_IF
(*
febInvalidProcessStep(CLK:=bInvalidProcessStepErrHold , Q=> );
*)
rebInvalidProcessStep(CLK:=bInvalidProcessStepErrHold AND bCallSt , Q=> );

IF rebInvalidProcessStep.Q THEN
bInvalidProcessStepErrPulse := TRUE;
END_IF


tInvalidProcessStepErrTimer(IN:= bInvalidProcessStepErrPulse , PT:=t#0.5s , Q=> , ET=> );

IF tInvalidProcessStepErrTimer.Q OR NOT bCallSt THEN
bInvalidProcessStepErrPulse := FALSE;
END_IF

(*Sequence Start*)
(*
IF NOT bSequenceSt THEN
iSeqStep := 0;
END_IF
*)
rebCallSt(CLK:=bCallSt , Q=> );
IF rebCallSt.Q (*OR (CallSelfCheckRE.Q*) AND NOT bInvalidProcessStepErrHold(*) OR febInvalidProcessStep.Q*) THEN
iSeqStep := 1;
(*iCurrentProcessStep := 1;*)
END_IF

rebInvalidStnSeqRepCall(CLK:=DSStnSeqRepCall.bInvalidCallStationSequenceNoPulse , Q=> );
rebInvalidStnSubRepCall(CLK:=DSStnSeqSubCall.bInvalidCallSubRecipeNoPulse , Q=> );


CASE iSeqStep OF

0:;

1: (*Select Sequence Recipe By Refering Basket Information*)
bCallStnSeqRecipeErr := FALSE;
bCallStnSubRecipeErr := FALSE;

DSStnSeqRepCall.Call_iStationSequenceRecipe := DSBasketInfo.iStationSeqenceRecipeNo(*iProgramNo*);
DSStnSeqRepCall.bCallPB := TRUE;

IF DSStnSeqRepCall.bCallCompleted THEN
DSStnSeqRepCall.bCallPB := FALSE;

iSeqStep:=2;

END_IF

IF rebInvalidStnSeqRepCall.Q THEN
DSStnSeqRepCall.bCallPB := FALSE;

iSeqStep:=11;
END_IF



2: (*Select Sub Recipe By Refering Selected Sequence Recipe Number*)

DSStnSeqSubCall.Call_iSubRecipe := DSStnSeqRepCall.Call_DsStationSequenceRecipeMemory.AR10iStationSubProNo[iCurrentProcessStep];
DSStnSeqSubCall.bCallPB := TRUE;


IF DSStnSeqSubCall.bCallCompleted THEN
DSStnSeqSubCall.bCallPB := FALSE;

iSeqStep:=3;
END_IF

IF rebInvalidStnSubRepCall.Q THEN
DSStnSeqSubCall.bCallPB := FALSE;

iSeqStep:=12;
END_IF


3: (*Transfer Sub Recipe Detail to Buffer*)

	BuffersSubDescription := DSStnSeqSubCall.Call_sSubDescription ;
	BufferDsSubRecipeMemory := DSStnSeqSubCall.Call_DsSubRecipeMemory;

iPreviousProcessStep := iCurrentProcessStep;
bCallCompleted := TRUE;
CallSelfCheckHR := FALSE;
iSeqStep:=4;

4:

CallCompletedTimer(IN:= bCallCompleted , PT:=t#0.5s , Q=> , ET=> );

IF CallCompletedTimer.Q THEN
bCallCompleted := FALSE;
END_IF


11:
iPreviousProcessStep := iCurrentProcessStep;
CallSelfCheckHR := FALSE;
bCallStnSeqRecipeErr := TRUE;
iSeqStep:=21;

12:
iPreviousProcessStep := iCurrentProcessStep;
bCallStnSubRecipeErr := TRUE;
CallSelfCheckHR := FALSE;
iSeqStep:=22;

21:;

22:;


END_CASE

END_FUNCTION_BLOCK

// ---- FBs/B_JKS_NewFB_V2/FBP-Memory_Sub/fbV2_GnrStationMasterController.TcPOU
FUNCTION_BLOCK fbV2_GnrStationMasterController

(*20171025 - Edit by Lim*)
(*Rung 337 - "bTransferStationBasketAvailable" variable control to solve the problem if for the basket can pick and tranfer to the same station*)


VAR_INPUT
	bTrackerEN								: BOOL;
	bTrackerBasedOnPreviousTime			: BOOL;
	bProcessCompleteBasedMasterTime		: BOOL;
	bBasketTransferCallArmInterlock			: BOOL; (* Temporary -> for GPM Only*)
	bReset									: BOOL;
	iCurrentStationAddress 					: INT;															(* Input - Define current station no so that this fb know which array number to used*)
	iPreCallArmTime							: INT;															(* Input - Pre-Call Arm Time, Program will call arm if the Total process timeEV Equal or Lesser than this value*)
	iTotalProcessTimeSV						:INT;
	iCurrentStnSeqProcessTotalTime 		: INT;															(* Input - Link with fbStnSeqProcess, to collect CurrentProcessTotalTime*)
	iPreviousStnSeqProcessTotalTime 		: INT; 															(* Input - Link with fbStnSeqProcess,  to collect PreviousProcessTotalTime*)
	iNonStopCurrentProcessTime: INT;
	bStnSeqProcessInProgressFlag			: BOOL;														(* Input - Link with fbStnSeqProcess,  to collect the status of process in progress from StnSeqProcessfb*)
	bStnSeqProcessCompleted 				: BOOL;														(* Input - Link with fbStnSeqProcess,  to collect the status of process completion from StnSeqProcessfb*)
	ARbAlternateStnEn : ARRAY [1..iAlternateSetQty] OF BOOL;
	AR2siAlternateStn : ARRAY [1..iAlternateSetQty, 1..iAlternateStnQty] OF INT;
(*	DSStnSeqProOutput 				:DS_StnSeqProOutput;								(* Output - To Control Output - When process running, instrument should control by the output in this Data structure*)
*)

END_VAR

VAR_IN_OUT PERSISTENT
	bStnSeqProcessSt						: BOOL;														(* Output - Link with fbStnSeqProcess, After Read out from fbGnrProductRecipeMemory, this fb will trigger this Bool to start the StnSeqProcess*)

	ARbProductRecipeCallEn 				: ARRAY [0..iStnQty] OF BOOL;					(* Output - Link with fbGnrProductRecipeMemory, Array based on Current Station No, the fbGnrProductRecipeMemory will start Read info from Memory when this bool turn on*)
	ARiProductRecipeNoCall 				: ARRAY [0..iStnQty] OF INT;						(* Output - Link with fbGnrProductRecipeMemory, Array based on Current Station No, the read out from fbGnrProductRecipeMemory is based on this Product Recipe No*)
	ARiProductRecipeStepCall 				: ARRAY [0..iStnQty] OF INT;						(* Output - Link with fbGnrProductRecipeMemory, Array based on Current Station No, the read out from fbGnrProductRecipeMemory is based on this Product Recipe Step No*)
	DSfbGnrProductRecipeMemoryOut 		: DSV2_fbGnrProductRecipeMemoryOut;						(* Input - Link with fbGnrProductRecipeMemory, all the read out info from fbGnrProductRecipeMemory will store in this DataStucture*)

	ARbArmReady						: ARRAY [1..iArmQty] OF BOOL;								(* Input - From ArmPnpFB, This signal is used to confirm if the arm is ready and idling*)
	ARiStnNoToCalledArm					: ARRAY [0..iArmQty] OF INT; 									(* Output - Link with fbArmPnP, Array based on Arm No, The Int will store which Station that calling the Arm*)
	ARDSGnrFeedArmPnpParameter		: ARRAY [0..iArmQty] OF DSV2_Gnr_CalledArmPnpParameter; 	(* Output - Link with fbArmPnP, Array based on Current Station No, Arm should move based on this DataStructure Info*)

	ARDSLdBasketInfo		 				: ARRAY [0..iLdStnQty] OF DSV2_BasketInfo;								(*Input - Loading CONFIRM Basket Info*)
	ARDSUldBasketInfo		 				: ARRAY [0..iUldStnQty] OF DSV2_BasketInfo;							(*Input - Uloading CONFIRM Basket Info*)
	ARDsStnBasketInfo					: ARRAY [0..iStnQty] OF DSV2_BasketInfo;									(*Input - Station Basket Info*)


END_VAR

VAR_OUTPUT PERSISTENT

	DSGnrBufferCalledArmPnpParameter 	: DSV2_Gnr_CalledArmPnpParameter;							(* Internal used, Buffer Data Structure read out from fbGnrProductRecipeMemory*)
	DSGnrBuffersPnpSequenceDescription	: STRING (99);													(* Internal used, Buffer Description read out from fbGnrProductRecipeMemory*)
	ARiPreviousStnSeqTotalProcessTime 	: ARRAY [0..iProductRecipeArrayQty] OF INT;				(* Internal used, Previous Total Process Time will save into this Array, Array based on StationSequenceNo*)
	iMasterTimeCallArmCountDownTime: INT;
	iMasterTimeBasedProcessCompleteFlag : BOOL;
	iCallStep									: INT;															(* Internal used, to monitor the current Step so that you can indentify the error of this function block if stucked*)

END_VAR
VAR PERSISTENT
	DSfbGnrProductRecipeMemoryOutErrorLog 		: DSV2_fbGnrProductRecipeMemoryOut;
	DSCurrentStationBasketInfoErrorLog				: DSV2_BasketInfo;

	bBasketDetectedRE						: R_TRIG;
	iCallCheck								: INT;
	bArmPnpSequenceCallEn				: BOOL;
	bStnSeqProcessCompletedRE			: R_TRIG;
	iCallArmCountDownTime				: INT;
	bCallArmEnInt								: BOOL;


END_VAR
VAR
	bBasketDetectedFE						: F_TRIG;
	bCallProductRecipeStorageEn			: BOOL;
	bTestCallArm								: BOOL;

	DSCurrentStationBasketInfo: DSV2_BasketInfo;
	DSEmptyBasketInfo: DSV2_BasketInfo;
	bPickStationBasketAvailable: BOOL;
	bTransferStationBasketAvailable: BOOL;
	bTransferStationBasketNotAvailable: BOOL;
	iCurrentStationAddressInt: INT;
	iTrackerCallArmCountDownTime: INT;
(*	bAlternateStnEnableFound: BOOL;*)
(*	iCheckAlternateStnEnFL: INT;*)
	bPickAltStnIDFound: BOOL;
	iPickAlternateStnFindFL: INT;
	iPickAlternateSetFindFL: INT;
	iPickAltStnTransferFL : INT;
	ARiBufferPickAltStn: ARRAY [1..iAlternateStnQty] OF INT;

	bTransferAltStnIDFound: BOOL;
	iTransferAlternateStnFindFL: INT;
	iTransferAlternateSetFindFL: INT;
	iTransferAltStnTransferFL : INT;
	ARiBufferTransferAltStn: ARRAY [1..iAlternateStnQty] OF INT;

	iCheckTrfStnBktFL: INT;
	iTransferStnNo: INT;
	iAltTransferStnNo: INT;
	iSearchLdStnFL: INT;
	bLdStnFound: BOOL;
	iSearchStnIDFL: INT;
	iSearchStnIDFound: BOOL;
	DSUldBasketInfo: BOOL;
	iSearchLdStnIDFound: BOOL;
	iSearchUldStnIDFound: BOOL;
	iCheckTrfStnBktSFL: INT;
	bReadyToCallArm: BOOL;
	bTrackerBasedPreviousTimeCallArm: BOOL;
	bTrackerNotBasedPreviousTimeCallArm: BOOL;
	bDataInBufferCalledArmPnpParameterDone: BOOL;
	bResetRE: R_TRIG;
	tErrorLoopingTimer: TON;
END_VAR

bResetRE(CLK:=bReset , Q=> );


(*Check if Loading Stn Detected, Switch the CurrentStatonAddress to 0*)
bLdStnFound:=FALSE;
iSearchLdStnFL := 1;
	FOR iSearchLdStnFL := 1 TO iLdStnQty DO
		IF iSearchLdStnFL >= 1 AND iSearchLdStnFL <= iLdStnQty THEN
			IF ARiLdStnID[iSearchLdStnFL] = iCurrentStationAddress THEN
			iCurrentStationAddressInt := 0;
			bLdStnFound:=TRUE;
			END_IF
		END_IF
	END_FOR

IF NOT bLdStnFound THEN
iCurrentStationAddressInt := iCurrentStationAddress;
END_IF


(*Check if Alternate Stn Matched with Current (Pick) Station*)
bPickAltStnIDFound := FALSE;
iPickAlternateSetFindFL := 1;
	FOR iPickAlternateSetFindFL := 1 TO iAlternateSetQty DO
		IF iPickAlternateSetFindFL >= 1 AND iPickAlternateSetFindFL <= iAlternateSetQty THEN
			IF ARbAlternateStnEn[iPickAlternateSetFindFL] THEN
			iPickAlternateStnFindFL := 1; (*Find Stn ID matching*)
				FOR iPickAlternateStnFindFL := 1 TO iAlternateStnQty DO
					IF iPickAlternateStnFindFL >= 1 AND iPickAlternateStnFindFL <= iAlternateStnQty THEN
						IF iCurrentStationAddress = AR2SiAlternateStn[iPickAlternateSetFindFL , iPickAlternateStnFindFL] THEN
							bPickAltStnIDFound := TRUE;
							iPickAltStnTransferFL := 1;
								FOR iPickAltStnTransferFL := 1 TO iAlternateStnQty DO
									IF iPickAltStnTransferFL >= 1 AND iPickAltStnTransferFL <= iAlternateStnQty THEN
										ARiBufferPickAltStn[iPickAltStnTransferFL] := AR2SiAlternateStn[iPickAlternateSetFindFL , iPickAltStnTransferFL];
									END_IF
								END_FOR
							iPickAlternateSetFindFL := iAlternateSetQty+1;
							iPickAlternateStnFindFL := iAlternateStnQty+1;
							iPickAltStnTransferFL := iAlternateStnQty+1;

						END_IF
					END_IF
				END_FOR
			END_IF
		END_IF
	END_FOR

(*Check if Alternate Stn Matched with Transfer Station*)

bTransferAltStnIDFound := FALSE;
IF iCallStep = 3 THEN
iTransferAlternateSetFindFL := 1;
	FOR iTransferAlternateSetFindFL := 1 TO iAlternateSetQty DO
		IF iTransferAlternateSetFindFL >= 1 AND iTransferAlternateSetFindFL <= iAlternateSetQty THEN
			IF ARbAlternateStnEn[iTransferAlternateSetFindFL] THEN
			iTransferAlternateStnFindFL := 1; (*Find Stn ID matching*)
				FOR iTransferAlternateStnFindFL := 1 TO iAlternateStnQty DO
					IF iTransferAlternateStnFindFL >= 1 AND iTransferAlternateStnFindFL <= iAlternateStnQty THEN
						IF DSGnrBufferCalledArmPnpParameter.iTransferStationNo = AR2SiAlternateStn[iTransferAlternateSetFindFL , iTransferAlternateStnFindFL] THEN
							bTransferAltStnIDFound := TRUE;
							iTransferAltStnTransferFL := 1;
								FOR iTransferAltStnTransferFL := 1 TO iAlternateStnQty DO
									IF iTransferAltStnTransferFL >= 1 AND iTransferAltStnTransferFL <= iAlternateStnQty THEN
										ARiBufferTransferAltStn[iTransferAltStnTransferFL] := AR2SiAlternateStn[iTransferAlternateSetFindFL , iTransferAltStnTransferFL];
									END_IF
								END_FOR
							iTransferAlternateSetFindFL := iAlternateSetQty+1;
							iTransferAlternateStnFindFL := iAlternateStnQty+1;
							iTransferAltStnTransferFL := iAlternateStnQty+1;

						END_IF
					END_IF
				END_FOR
			END_IF
		END_IF
	END_FOR
END_IF

(*Define Current Station Basket Info*)
iSearchLdStnIDFound := FALSE;
iSearchUldStnIDFound := FALSE;


IF NOT iSearchLdStnIDFound AND NOT iSearchUldStnIDFound THEN
	iSearchStnIDFL := 1;
		FOR iSearchStnIDFL := 1 TO iLdStnQty DO
			IF iSearchStnIDFL >= 1 AND iSearchStnIDFL <= iLdStnQty THEN
				IF iCurrentStationAddress = ARiLdStnID[iSearchStnIDFL] THEN
					DSCurrentStationBasketInfo := ARDSLdBasketInfo[iSearchStnIDFL];
					iSearchLdStnIDFound := TRUE;
				END_IF
			END_IF
		END_FOR
END_IF


IF NOT iSearchLdStnIDFound AND NOT iSearchUldStnIDFound THEN
	iSearchStnIDFL := 1;
		FOR iSearchStnIDFL := 1 TO iUldStnQty DO
			IF iSearchStnIDFL >= 1 AND iSearchStnIDFL <= iUldStnQty THEN
				IF iCurrentStationAddress = ARiUldStnID[iSearchStnIDFL] THEN
					DSCurrentStationBasketInfo := ARDSUldBasketInfo[iSearchStnIDFL];
					iSearchUldStnIDFound := TRUE;
				END_IF
			END_IF
		END_FOR
END_IF


IF NOT iSearchLdStnIDFound AND NOT iSearchUldStnIDFound THEN
	IF iCurrentStationAddress >= 1 AND iCurrentStationAddress <= iStnQty THEN
	DSCurrentStationBasketInfo := ARDsStnBasketInfo[iCurrentStationAddress];
	ELSE
	DSCurrentStationBasketInfo := DSEmptyBasketInfo;
	END_IF
END_IF


(* Check if no one called Data From DSfbGnrProductRecipeMemory *)
iCallCheck := 1;
FOR iCallCheck := 1 TO iStnQty DO
		IF ARbProductRecipeCallEn[iCallCheck] THEN
		bArmPnpSequenceCallEn := TRUE;
		iCallCheck := 90;
		END_IF
END_FOR

IF iCallCheck > iStnQty AND iCallCheck <= (iStnQty+2) THEN
bArmPnpSequenceCallEn := FALSE;
END_IF


